Omron CX-Programmer project PAGODE (CX-Programmer 9.42)
; PLC1-GROND ; PLC2-GROND  ;PLC3-EILAND

# PLC PLC1_PAGODE: CS1G-H CPU42

## Global symbols (name address type ; comment)
ALM_1152_PLC2 H172.00 BOOL  ; ALARM PLC 2 WAARDE ACT-SOLL TE GROOT
ALM_EIL_BYPASS W226.15 BOOL  ; STAB EILAND IN BYPASS
ANA_OUT_2_REAL D5420 REAL  ; ANALOG OUTPUT 2 REAL 4-20mA
ANA_OUT_2_SCALER D5418 REAL  ; ANALOG OUTPUT 2 SCALER FOR 4-20mA
ARM_MOTION_PULSE 0142 NUMBER  ; ARM MOTION PULSER
ARM_POSITION_VALUE_ANA_OUT D5430 INT  ; ARM POSITION VALUE TO ANALOG OUTPUT
ARM_SPEED D5522 REAL  ; ARM SPEED IN DEGREE PER MINUTE
ARM_SPEED_FILTERED D6020 REAL  ; ARM SPEED FILTERED IN DEGREE PER MINUTE
ARM_SPEED_FILTER_01 D6000 REAL  ; ARM SPEED FILTER 01
ARM_SPEED_FILTER_02 D6002 REAL  ; ARM SPEED FILTER 01
ARM_SPEED_FILTER_03 D6004 REAL  ; ARM SPEED FILTER 03
ARM_SPEED_FILTER_04 D6006 REAL  ; ARM SPEED FILTER 04
ARM_SPEED_FILTER_05 D6008 REAL  ; ARM SPEED FILTER 05
ARM_SPEED_RESULT_01 D6010 REAL  ; RESULT 01
ARM_SPEED_RESULT_02 D6012 REAL  ; RESULT 02
ARM_SPEED_RESULT_03 D6014 REAL  ; RESULT 03
ARM_SPEED_RESULT_04 D6016 REAL  ; RESULT 04
Act_Snelheid_Aansturing_Arm D177 INT  ; Actuele snelheid aansturing Arm
1527.00 BOOL  ; Controllink Node 1 online
1527.01 BOOL  ; Controllink Node 2 online
1527.02 BOOL  ; Controllink Node 3 Online
2020.00 BOOL  ; COUNT
3012.02 BOOL  ; stop vanaf grond
3034.06 BOOL  ; COMMUNICATIE PLC 1 NAAR PLC 2 HYDRAULIEK UNIT ARM INBEDRIJF
3327.00 BOOL  ; Ingangspoort rechts gesloten Van PLC 2
3327.01 BOOL  ; Inganspoort links gesloten van PLC2
3337.03 BOOL  ; One Shot Pulse t.b.v. ramp tijd
56.05 BOOL  ; stop show
D1200 CHANNEL  ; SIMPLE COUNTER MODE
D1202 CHANNEL  ; COUNTER 2
D134 CHANNEL  ; help_abs_enc1
D190 CHANNEL  ; encoder_4_1
D191 CHANNEL  ; ecoder_4_2
D20 CHANNEL  ; `
H102.01 BOOL  ; Controllink Node 1 offline (PLC 1)
H102.02 BOOL  ; Controllink Node 2 offline (PLC 2)
H102.03 BOOL  ; Controllink Node 3 offline (PLC 3)
H102.05 BOOL  ; Algemene storing voor Controllink unit.
H102.06 BOOL  ; Storing Controllink Node 1
H102.07 BOOL  ; Storing Controllink Node 2
H102.08 BOOL  ; Storing Controllink Node 3
H121.03 BOOL  ; UPS in storing of batterijbedrijf
H121.04 BOOL  ; Alarm 1-0340 Hoge temperatuur in Technische Ruimte Pagode.
H158.09 BOOL  ; $?St$Bk?_#[29956] / Benedenpositie eiland wijkt af van encoder positie (42S10) / $?St$Bk?_#[29956]
H158.10 BOOL  ; $?St$Bk?_#[29957] / Ondermelding eiland niet binnen encoder waarden (41S4) / $?St$Bk?_#[29957]
H158.11 BOOL  ; $?St$Bk?_#[29958] / Ondermelding eiland niet binnen encoder waarden (41S7) / $?St$Bk?_#[29958]
H186.01 BOOL  ; $?St$Bk?_#[29959] / Alarm 1 - 1377 Poort 1 Links. Pal niet gevallen / $?St$Bk?_#[29959]
H186.02 BOOL  ; Alarm 1 - 1378 Poort 1 Links. Open sensor schakeld ongewenst. ( )
H186.03 BOOL  ; Alarm 1 - 1379 Poort 1 Links. Open sensor schakeld niet ( )
H186.04 BOOL  ; $?St$Bk?_#[29960] / Alarm 1 - 1380 Poort 1 Links. Bijna open sensor schakeld ongewenst. ( ) / $?St$Bk?_#[29960]
H186.05 BOOL  ; Alarm 1 - 1381 Poort 1 Links. Bijna open sensor schakeld niet ( )
H186.06 BOOL  ; Alarm 1 - 1382 Poort 1 Links. Sluit sensor schakeld ongewenst. ( )
H186.07 BOOL  ; Alarm 1 - 1383 Poort 1 Links. Sluit sensor schakeld niet ( )
H186.08 BOOL  ; $?St$Bk?_#[29961] / Alarm 1 - 1384 Poort 1 Links. Beknelling bewaking aangesproken. ( ) / $?St$Bk?_#[29961]
H400 CHANNEL  ; Algemene alarmen PLC 3 draaiend deel eiland
H401 CHANNEL  ; Alarmen Ingangspoort Links 1
H401.00 BOOL  ; $?St$Bk?_#[29962] / Alarm 1 - 1376 Poort 1 Links. Pal meldt niet omhoog / $?St$Bk?_#[29962]
H402 CHANNEL  ; Alarmen Ingangspoort Links 2
H403 CHANNEL  ; Alarmen Ingangspoort Rechts 1
H404 CHANNEL  ; Alarmen Ingangspoort Rechts 2
H405 CHANNEL  ; Alarmen Uitgangspoort Links 1
H406 CHANNEL  ; Alarmen Uitgangspoort Links 2
H407 CHANNEL  ; Alarmen Uitgangspoort Rechts 1
H408 CHANNEL  ; Alarmen Uitgangspoort Rechts 2
T0141 BOOL  ; DELAY ARM STAR
T0142 BOOL  ; ARM MOTION PULSER
T0150 BOOL  ; TIMER ENCODER 1 FAUT
T0151 BOOL  ; TIMER ENCODER 2 FAULT
T0198 BOOL  ; Delay Eiland op positie (1.04)
T0224 BOOL  ; ALARM 1-1454 SIGNAL STATUS VALVE 145 NOT OK
T0225 BOOL  ; ALARM 1-1455 OIL LEVEL 2 NOT OK
T0230 BOOL  ; ALARM 1-1462 HARDWARE WATCHDOG FROM HAGENBUCH MISSING TIMER ON
T0231 BOOL  ; ALARM 1-1462 HARDWARE WATCHDOG FROM HAGENBUCH MISSING TIMER OFF
T0240 BOOL  ; TIMER ARM HYDRAULIC ON
T0241 BOOL  ; TIMER ISLAND HYDRAULIC ON
T0310 BOOL  ; TIMER RESET ERROR HAGENBUCH SYSTEM
T0311 BOOL  ; PRESET INCLINOMETER HAGENBUCH
T0320 BOOL  ; Timer Alarm 1191
T0321 BOOL  ; Timer Alarm 1192
T0661 BOOL  ; \
W160.04 BOOL  ; blok_tourn
W160.06 BOOL  ; blokkeer_links
W160.07 BOOL  ; blokkeer_rechts
W20.03 BOOL  ; Merker Watchdog Communicatie OK Plc 1 & Plc 2
W231.15 BOOL  ; EILAND ROND GEWEEST
W56.03 BOOL  ; hydrau
W56.05 BOOL  ; stop show van grond
W56.06 BOOL  ; stop show van eiland
W90.00 BOOL  ; Blokkeer Tourniquet
W90.01 BOOL  ; Verhoog aantal
W90.02 BOOL  ; Blokkeer tourniquet links
W91.00 BOOL  ; Blokkeer Tourniquet
W91.01 BOOL  ; Verhoog aantal
W91.02 BOOL  ; Blokkeer tourniquet rechts
BT_Hydr_Main_Pump_Arm_On T0194 BOOL  ; Hydraulic main pump arm on delay timer
BT_MS_11Q08_not_OK T0195 BOOL  ; Hydraulic main pump arm MS 11Q08 not OK
BT_MS_11Q10_not_OK T0196 BOOL  ; Hydraulic main pump arm MS 11Q10 not OK
BT_MS_11Q12_not_OK T0197 BOOL  ; Hydraulic main pump arm MS 11Q12 not OK
COM1_AKTIEF_ALARM 3006.00 BOOL
COM1_ARM_ENAB_NEER 3024.03 BOOL  ; ARM ENABLE OMLAAG  VANUIT CYCLUS
COM1_ARM_OMHOOG 3037.00 BOOL  ; PLC 1 ARM OMHOOG
COM1_ARM_OMLAAG 3037.01 BOOL  ; PLC   1 ARM OMLAAG
COM1_ING_L_SLUITEN 3032.04 BOOL  ; VERZOEK SLUITEN INGANGS POORT LINKS
COM1_ING_R_OPEN 3032.05 BOOL  ; VERZOEK OPENEN INGANGS POORT RECHTS
COM1_ING_R_SLUITEN 3032.06 BOOL  ; VERZOEK SLUITEN INGANGS POORT RECHTS
COM1_Noodstop_Vertraagt_PLC1_OK 3004.04 BOOL  ; Communicatie Noodstop Vertaagt Plc 1 Ok Plc 1 naar Plc 2
COM1_STAPWOORD 3023 CHANNEL  ; STAP WOORD
COM1_TOURN_R 3031.01 BOOL  ; VERZOEK ENABLE TOURNIKET RECHTS
COM2_AKTIEF_ALARM 3306.00 BOOL
COM2_ARM_ENAB_NEER 3324.02 BOOL  ; ARM ENABLE OMLAAG VANUIT CYCLUS
COM2_ARM_ENAB_OP 3324.01 BOOL  ; ARM ENABLE OMHOOG VANUIT CYCLUS
COM2_ARM_OMHOOG 3337.00 BOOL  ; PLC 2 ARM OMHOOG
COM2_ARM_OMLAAG 3337.01 BOOL  ; PLC 2 ARM OMLAAG
COM2_ARM_SLOW 3324.05 BOOL  ; EILAND SLOW
COM2_CYCLUS_ENABLE 3324.15 BOOL  ; CYCLUS ENABLE
COM2_CYCLUS_STOP 3324.14 BOOL  ; VOORTIJDIGE STOP
COM2_EIL_STAB 3324.04 BOOL  ; EILAND STABILISATIE
COM2_ENAB_TOURNIKET 3324.10 BOOL  ; ENABLE TOURNIKET
COM2_ING_L_OPEN 3332.03 BOOL  ; VRIJGAVE INGANGS POORTEN L OPENEN VAN PLC 2
COM2_ING_L_SLUITEN 3332.04 BOOL  ; VRIJGAVE SLUITEN INGANGS POORT L VAN PLC 2
COM2_ING_R_OPEN 3332.05 BOOL  ; VRIJGAVE OPENEN INGANGS POORTEN RECHTS
COM2_ING_R_SLUITEN 3332.06 BOOL  ; VRIJGAVE SLUITEN INGANGS POORT RECHTS VAN PLC 2
COM2_LADING_WISSEL 3324.12 BOOL  ; BELADING EILAND WISSELEN
COM2_PB_EXIT_GATE 3033.00 BOOL  ; PUSH BUTTON EXIT GATE FROM ISLAND (PLC3)
COM2_POORT_DICHT 3324.09 BOOL  ; ALLE POORTEN GESLOTEN
COM2_POORT_ENAB 3324.00 BOOL  ; POORT ENABLE VANUIT CYCLUS
COM2_READY_START 3324.13 BOOL  ; READY VOOR START
COM2_RIDE_HOME 3324.11 BOOL  ; RIDE HOME
COM2_ROTATIE 3324.03 BOOL  ; ROTATIE ENABLE VANUIT CYCLUS
COM2_STAP0 3323.00 BOOL  ; STAP 0 CYCLUS
COM2_STAP1 3323.01 BOOL  ; STAP 1 CYCLUS
COM2_STAP10 3323.10 BOOL  ; STAP 10 CYCLUS
COM2_STAP13 3323.13 BOOL  ; STAP 13 CYCLUS
COM2_STAP14 3323.14 BOOL  ; STAP 14 CYCLUS
COM2_STAP15 3323.15 BOOL  ; STAP 15 CYCLUS
COM2_STAP2 3323.02 BOOL  ; STAP 2 CYCLUS
COM2_STAP3 3323.03 BOOL  ; STAP 3 CYCLUS
COM2_STAP4 3323.04 BOOL  ; STAP 4 CYCLUS
COM2_STAP5 3323.05 BOOL  ; STAP 5 CYCLUS
COM2_STAP6 3323.06 BOOL  ; STAP 6 CYCLUS
COM2_STAP7 3323.07 BOOL  ; STAP 7 CYCLUS
COM2_STAP8 3323.08 BOOL  ; STAP 8 CYCLUS
COM2_STAP9 3323.09 BOOL  ; STAP 9 CYCLUS
COM2_STAPWOORD 3323 CHANNEL  ; STAP WOORD
COM2_TOURN_L 3331.00 BOOL  ; TOESTEMMING VRIJG TOURNIKET L
COM2_TOURN_R 3331.01 BOOL  ; TOESTEMMING VRIGAVE TOURNIKET RECHTS
COM_TOURN_R 562.01 BOOL  ; VERZOEK VRIJGAVE TOURNIKET R
COUNTER_RESET_CH_1 2020.04 BOOL  ; COUNTER RESET CHANNEL 1
COUNTER_RESET_CH_2 2020.05 BOOL  ; COUNTER RESET CHANNEL 2
COUNT_CARD_CH1_INI D20201 CHANNEL  ; COUNTER CARD CHANNEL 1 INITIALISATION
COUNT_CARD_GEN_INI D20200 CHANNEL  ; COUNTER CARD GENERAL INITIALISATION
COUNT_GEN_ENABLE 2020.00 BOOL  ; COUNTERS GENERAL ENABLE
COUT_CARD_CH2_INI D20202 CHANNEL  ; COUNTER CARD CHANNEL 2 INITIALISATION
C_CONTROL D108 UINT  ; CONTROL BCD NAAR BIN COUNTERS
Com1_3_Eiland_Poortjes_Gesloten 906.00 BOOL  ; Merker Eiland Poortjes zijn Gesloten
Com1_3_Lamp_Ingangs_Poortjes_Geopend_Eiland 902.02 BOOL  ; Communicatie Lampje (16H2) Ingangs Poortje s 1 + 2 Geopend Eiland Plc 1 & Plc 2 naar Plc 3
Com1_3_Lamp_Ready_For_Dispatch 902.01 BOOL  ; Communicatie Ready for Dispatch Lampje Eiland (16H2) Plc 1 & Plc 2 naar Plc 3
Com1_3_Vrijgave_Poortjes_Eiland 906.01 BOOL  ; Communicatie Vrijgave Eiland Poortjes Plc 1 & Plc 2 naar Plc 3
Com1_44HS12 3011.15 BOOL
Com1_44HS14 3012.00 BOOL
Com1_91H10 3011.04 BOOL  ; Communicatie Lampje Algemeen Alarm Plc 1 naar Plc 2
Com1_91H12 3011.05 BOOL  ; Communicatie Lampje Show Plc 1 naar Plc 2
Com1_91H14 3011.06 BOOL  ; Communicatie Lampje Linkse Tourniquet Ontgrendelt Plc 1 naar Plc 2
Com1_91H16 3011.07 BOOL  ; Communicatie Lampje Rechtse Tourniquet Ontgrendelt Plc 1 naar Plc 2
Com1_91H18 3011.08 BOOL  ; Communicatie Lampje Arm & Eiland Omhoog Plc 1 naar Plc 2
Com1_91H2 3011.00 BOOL  ; Communicatie Lampje Sturrspanning Ingeschakeld Plc 1 naar Plc 2
Com1_91H4 3011.01 BOOL  ; Communicatei Lampje Handbedrijf Ingeschakeld Plc 1 naar Plc2
Com1_91H6 3011.02 BOOL  ; Communicatie Lampje Automatisch bedrijf Ingeschakeld Plc 1 naar Plc 2
Com1_91H8 3011.03 BOOL  ; Communicatie Lampje Pompen in Bedrijf Plc 1 naar Plc 2
Com1_92H12 3011.14 BOOL
Com1_92H2 3011.09 BOOL  ; Communicatie Lampje Arm & Eiland Omlaag Plc 1 naar Plc 2
Com1_92H4 3011.10 BOOL  ; Communicatie Lampje Rotatie Eiland Linksom Plc 1 naar Plc 2
Com1_92H6 3011.11 BOOL  ; Communicatie Lampje Rotatie Eiland Rechtsom Plc 1 naar Plc 2
Com1_92H8 3011.12 BOOL  ; Service schakelaar technische dients
Com1_92S14 3011.15 BOOL
Com1_92Z10 3011.13 BOOL
Com1_Act_Groter_Snelheid 3037.04 BOOL  ; Actuele snelheid groter dan wens snelheid
Com1_Act_Kleiner_Snelheid 3037.06 BOOL  ; Actuele snelheid kleiner dan wens snelheid
Com1_Act_gelijk_Snelheid 3037.05 BOOL  ; Actuele snelheid gelijk aan de wens snelheid
Com1_Arm_Home 3024.01 BOOL  ; Arm is geheel beneden
Com1_Arm_Omhoog 3037.01 BOOL  ; PLC 1 ARM OMHOOG
Com1_Arm_Omlaag 3037.02 BOOL  ; PLC 1ARM OMLAAG
Com1_Auto_Bedrijf 3010.01 BOOL  ; Communicatie Auto Bedrijf van Plc 1 Naar Plc 2
Com1_Auto_Rotatie_Rechtsom 3047.02 BOOL
Com1_Auto_Rotatie_linksom 3047.01 BOOL  ; Communicatie Auto Rotatie Linksom
Com1_E_Stop_Niet_Gedrukt 3004.00 BOOL  ; Communicatie E-stop niet gedrukt Plc 1 naar Plc 2
Com1_Eiland_Poortjes_Gesloten 3044.00 BOOL  ; Communicatie Eiland Poortjes Gesloten Plc 1 naar Plc 2
Com1_Eiland_Rond_Geweest 3047.14 BOOL
Com1_Eiland_Stab_Linksom 3046.01 BOOL  ; Communicatie Plc 1 naar Plc 2 Stabiliseer het Eiland naar Links
Com1_Eiland_Stab_Rechtsom 3046.02 BOOL  ; Communicatie Plc 1 naar Plc 2 Stabiliseer het Eiland naar Rechts
Com1_Enable_Freq_Contr_Linksom 3047.13 BOOL
Com1_Enable_Freq_Contr_Rechtsom 3047.12 BOOL
Com1_Enable_Hydrau_Eiland 3045.00 BOOL  ; Communicatie Enable Hydrau Eiland Plc 1 naar Plc 2
Com1_Enable_Stabilisatie 3046.00 BOOL  ; Communicatie Plc 1 naar Plc 2 Enable de Eiland Stabilisatie
Com1_Hand_Bedrijf 3010.00 BOOL  ; Communicatie Hand Bedrijf Plc 1 naar plc 2
Com1_Hardw_Watchdogs_OK 3003.05 BOOL  ; Communicatie Plc 1 Watchdog plc 2 ok
Com1_Hardw_Watchdogs_ON 3003.04 BOOL  ; Communicatie Hardware Watchdog Plc 1 ON
Com1_Hoofd_Pomp_Hydrau_Grond 3034.02 BOOL  ; COMMUNICATIE PLC 1 NAAR PLC 2 START HOOFDPOMP HYDRAULIEK UNIT ARM
Com1_Hoofdpomp_Hydrau_Eiland 3045.03 BOOL  ; Communicatie Hoofdmotor Hydrau Eiland Aan Plc 1 naar Plc 2
Com1_Hoofdschakelaar_OK 3008.01 BOOL  ; Communicatie Hoofdschakelaar (3K7) OK (geen Kortsluiting of overbelasting)
Com1_Hydrau_Arm_OK 3034.06 BOOL  ; COMMUNICATIE PLC 1 NAAR PLC 2 HYDRAULIEK UNIT ARM INBEDRIJF
Com1_Hydrau_Eiland_ON 3045.01 BOOL  ; Communicatie Start Hydrau Pompen Plc 1 naar Plc 2
Com1_Hydrauliek_Eiland_Inbedrijf 3045.15 BOOL
Com1_Ingang_Poortje_1_L_Dicht 3032.02 BOOL  ; Communicatie Plc 1 naar Plc 2 Open Ingangs poortjes
Com1_Ingangs_Poortje_1_Links_Open 3032.01 BOOL
Com1_Ingangs_Poortjes_Gesloten 3032.07 BOOL
Com1_Inst_Autom_7F12_Eiland_OK 3008.13 BOOL  ; Communicatie Installatie-Automaat Eiland (7F12) OK Plc 1 naar Plc 2
Com1_Inst_Autom_7F3_Eiland_OK 3008.10 BOOL  ; Communicatie Installatie-Automaat Eiland (7F3) OK Plc 1 naar Plc 2
Com1_Inst_Autom_7F5_Eiland_OK 3008.11 BOOL  ; Communicatie Installatie-Automaat Eiland (7F5) OK Plc 1 naar Plc 2
Com1_Inst_Autom_7F7_Eiland_OK 3008.12 BOOL  ; Communicatie Installatie-Automaat Eiland (7F7) OK Plc 1 naar Plc 2
Com1_Inst_Autom_8F11_Eiland_OK 3008.15 BOOL  ; Communicatie Installatie-Automaat Eiland (8F11) OK Plc 1 naar Plc 2
Com1_Inst_Autom_8F14_Eiland_OK 3009.00 BOOL  ; Communicatie Installatie-Automaat Eiland (8F14) OK Plc 1 naar Plc 2
Com1_Inst_Autom_8F17_Eiland_OK 3009.01 BOOL  ; Communicatie Installatie-Automaat Eiland (8F17) OK Plc 1 naar Plc 2
Com1_Inst_Autom_8F3_Eiland_OK 3008.14 BOOL  ; Communicatie Installatie-Automaat Eiland (8F3) OK Plc 1 naar Plc 2
Com1_Inst_Automaat_7F3_OK 3008.02 BOOL  ; Communicatie Installatie-Automaat (7F3) OK Plc 1 naar Plc 2
Com1_Inst_Automaat_7F5_OK 3008.03 BOOL  ; Communicatie Installatie-Automaat (7F5) OK Plc 1 naar Plc 2
Com1_Inst_Automaat_7F7_OK 3008.04 BOOL  ; Communicatie Installatie-Automaat (7F7) OK Plc 1 naar Plc 2
Com1_Inst_Automaat_8F11_OK 3008.06 BOOL  ; Communicatie Installatie-Automaat (8F11) OK Plc 1 naar Plc 2
Com1_Inst_Automaat_8F13_OK 3008.07 BOOL  ; Communicatie Installatie-Automaat (8F13) OK Plc 1 naar Plc 2
Com1_Inst_Automaat_8F15_OK 3008.08 BOOL  ; Communicatie Installatie-Automaat (8F15) OK Plc 1 naar Plc 2
Com1_Inst_Automaat_8F3_OK 3008.05 BOOL  ; Communicatie Installatie-Automaat (8F3) OK Plc 1 naar Plc 2
Com1_Inst_Automaat_9F11_OK 3008.09 BOOL  ; Communicatie Installatie-Automaat (9F11) OK Plc 1 naar Plc 2
Com1_Koelingspomp_Hydrau_Arm 3034.03 BOOL  ; COMMUNICATIE PLC 1 NAAR PLC 2 START KOELER POMP HYDRAULIEK UNIT ARM
Com1_Lamp_Eiland_Ingangs_poortjes_Geopend 3013.02 BOOL  ; Communicatie Lampje (16H2) Ingangs Poortje s 1 + 2 Geopend Eiland Plc 1 naar Plc 2
Com1_Lamp_Eiland_Ingangs_poortjes_Gesloten 3013.03 BOOL  ; Communicatie Lampje (16H3) Ingangs Poortje s 1 + 2 Gesloten Eiland Plc 1 naar Plc 2
Com1_Lamp_Eiland_Uitgangs_poortjes_Geopend 3013.05 BOOL  ; Communicatie Lampje (16H4) Uitgangs Poortje s 1 + 2 Geopend Eiland Plc 1 naar Plc 2
Com1_Lamp_Ready_For_Dispatch 3013.01 BOOL  ; Communicatie Lampje (16H3) Ready For Dispatch Eiland Plc 1 naar Plc 2
Com1_Noodstop_Direct_PLC1_OK 3004.03 BOOL  ; Communicatie NoodStop Direct OK Plc 1 naar Plc 2
Com1_Noodstop_PLC_1_OK 3004.02 BOOL  ; Communicatie Noodstop Plc 1 OK
Com1_Open_Ingangs_Poort_1_L 3032.03 BOOL
Com1_Open_Uitgangs_Poortjes 3033.03 BOOL  ; Open de Uitgangs Poortjes
Com1_Power_Freq_Reg_4A1 3047.00 BOOL  ; Communicatie Frequentie Regelaar (4A1) Voeding (72K6) Plc 1 naar 2
Com1_Pulse 3037.03 BOOL
Com1_Ready_To_Start_Show 3024.07 BOOL  ; Ready to Start Show
Com1_Ready_to_Reset_E_Stop 3004.01 BOOL  ; Communicatie Ready om de Noodstop te Resetten Plc 1 naar Plc 2
Com1_Reinigingspomp_Hydrau_Arm 3034.04 BOOL  ; COMMUNICATIE PLC 1 NAAR PLC 2 START OLIE REINIGINGS POMP HYDRAULIEK UNIT ARM
Com1_Reset_Trigger 3037.07 BOOL
Com1_Rotatie_Linksom 3047.04 BOOL
Com1_Rotatie_Rechtsom 3047.08 BOOL
Com1_Rotatie_Snel_Linksom 3047.06 BOOL
Com1_Rotatie_Snel_Rechtsom 3047.10 BOOL
Com1_Rotatie_Traag_Linksom 3047.05 BOOL
Com1_Rotatie_Traag_Rechtsom 3047.09 BOOL
Com1_SK_Open_Linker_Ingangs_Poortje_Eiland 3014.09 BOOL
Com1_SK_Open_Linker_Ingangs_Poortje_Oever 3014.11 BOOL
Com1_SK_Open_Linker_Uitgangs_Poortjes_Eiland 3014.13 BOOL
Com1_SK_Open_Rechter_Ingangs_Poortje_Eiland 3014.10 BOOL
Com1_SK_Open_Rechter_Ingangs_Poortje_Oever 3014.12 BOOL
Com1_SK_Open_Rechter_Uitgangs_Poortje_Eiland 3014.14 BOOL
Com1_SK_Open_Sluit_Linker_Oever_Poortjes_ 3014.05 BOOL
Com1_SK_Open_Sluit_Rechter_Oever_Poortjes_ 3014.06 BOOL
Com1_SK_Open_Uitgangs_Poortjes_Oever 3014.15 BOOL
Com1_SK_Reset_Alarmen 3014.01 BOOL
Com1_SK_SPARE_3314_00 3014.00 BOOL
Com1_SK_SPARE_3314_02 3014.02 BOOL
Com1_SK_SPARE_3315_03 3015.02 BOOL
Com1_SK_SPARE_3315_07 3015.07 BOOL
Com1_SK_SPARE_3315_08 3015.08 BOOL
Com1_SK_SPARE_3315_09 3015.09 BOOL
Com1_SK_Stabilisatie_Eiland_Linksom 3015.05 BOOL
Com1_SK_Stabilisatie_Eiland_Rechtsom 3015.06 BOOL
Com1_SK_Start_Stop_Hoofdpomp_Arm 3015.01 BOOL
Com1_SK_Start_Stop_Hoofdpomp_Eiland 3015.04 BOOL
Com1_SK_Start_Stop_Hydrau 3014.03 BOOL
Com1_SK_Start_Stop_Show 3014.04 BOOL
Com1_SK_Start_Stop_Stuurpomp_Arm 3015.00 BOOL
Com1_SK_Start_Stop_Stuurpomp_Eiland 3015.03 BOOL
Com1_SK_Vrijgave_Linker_Tourniquet 3014.07 BOOL
Com1_SK_Vrijgave_Rechter_Tourniquet 3014.08 BOOL
Com1_SK_WCD_1 3015.10 BOOL
Com1_SK_WCD_2 3015.11 BOOL
Com1_SK_WCD_3 3015.12 BOOL
Com1_SK_WCD_4 3015.13 BOOL
Com1_SK_WCD_5 3015.14 BOOL
Com1_SK_WCD_6 3015.15 BOOL
Com1_Service_Bedrijf_Ch_A 3010.02 BOOL  ; Communicatie Service Bedrijf Channel A van Plc 1 Naar Plc 2
Com1_Service_Bedrijf_Ch_B 3010.03 BOOL  ; Communicatie Service Bedrijf Channel B van Plc 1 Naar Plc 2
Com1_Show_Afbreken 3024.04 BOOL  ; Show Afbreken
Com1_Show_Arm_Omhoog 3024.08 BOOL  ; Show Arm Omhoog
Com1_Show_Arm_Omlaag 3024.09 BOOL  ; Show Arm Omlaag
Com1_Show_Eiland_Rotatie 3024.11 BOOL  ; Show Eiland Rotatie
Com1_Show_Eiland_Stabilisatie 3024.10 BOOL  ; Show Eiland Stabilisatie
Com1_Show_Stap_0 3023.00 BOOL  ; Show Stap 0
Com1_Show_Stap_1 3023.01 BOOL  ; Show Stap 1
Com1_Show_Stap_10 3023.10 BOOL  ; Show Stap 10
Com1_Show_Stap_2 3023.02 BOOL  ; Show Stap 2
Com1_Show_Stap_4 3023.04 BOOL  ; Show Stap 4
Com1_Show_Stap_5 3023.05 BOOL  ; Show Stap 5
Com1_Show_Stap_6 3023.06 BOOL  ; Show Stap 6
Com1_Show_Stap_7 3023.07 BOOL  ; Show Stap 7
Com1_Show_Stap_8A 3023.11 BOOL  ; Show Stap 8 A
Com1_Show_Stap_8B 3023.12 BOOL  ; Show Stap 8 B
Com1_Show_Stap_9 3023.09 BOOL  ; Show Stap 9
Com1_Show_stap_8 3023.08 BOOL  ; Show Stap 8
Com1_Sluit_Uitgangs_Poortjes_Oever 3033.04 BOOL  ; Sluit de Uitgangs Poortjes Oever
Com1_Smeertoestel_Hydrau_Arm 3034.05 BOOL  ; COMMUNICATIE PLC 1 NAAR PLC 2 START SMEER TOESTEL HYDRAULIEK UNIT ARM
Com1_Softw_Watchdog_Plc_2_OK 3003.03 BOOL  ; Communicatie Software Watchdog Plc 2 OK
Com1_Softw_watchdog_Plc_1_on 3003.00 BOOL  ; Communicatie Plc 1 Watchdog plc 1 on
Com1_Softw_watchdog_Pulse_Plc_1 3003.01 BOOL  ; Communicatie Software Watchdog Pulse Plc 1
Com1_Spannings_Beveiliging_OK 3008.00 BOOL  ; Communicatie Onder- OverSpannings beveiliging OK
Com1_Stap_3 3023.03 BOOL  ; Show Stap 3
Com1_Stop_Show 3024.05 BOOL  ; Stop Show
Com1_Stuur_Pomp_Hydrau_Grond 3034.01 BOOL  ; VERZOEK  STUUR POMP HYDRAULIEK UNIT ARM
Com1_Stuurpomp_Hydrau_Arm 3034.01 BOOL  ; COMMUNICATIE PLC 1 NAAR PLC 2 START STUUR POMP HYDRAULIEK UNIT ARM
Com1_Stuurpomp_Hydrau_Eiland 3045.02 BOOL  ; Communicatie StuurPompen Aan Hydrualiek Eiland Plc 1 naar Plc 2
Com1_Tilt_switches_OK 3042.00 BOOL  ; Communicatie Tilt Switches OK Plc 1 naar Plc 2
Com1_Uitgangs_poortjes_Dicht 3033.02 BOOL  ; Uitgangs Poortjes zijn Gesloten
Com1_Uitgangs_poortjes_Open 3033.01 BOOL  ; Uitgangs Poortjes Zijn Open
Com1_VRIJGAVE_HYDRAU_ARM 3034.00 BOOL  ; COMMUNICATIE PLC 1 NAAR PLC 2 VRIJGAVE HYDRAULIEK UNIT ARM
Com1_Verhinder_Start_Show 3024.06 BOOL  ; Verhinder de Start van de Show
Com1_Vrijgave_Arm_Beweging 3037.00 BOOL
Com1_Vrijgave_Eiland_Poortjes 3044.01 BOOL  ; Communicatie Vrijgave Eiland Poortjes Plc 1 naar Plc 2
Com1_Vrijgave_Ingangs_Poortjes 3032.00 BOOL
Com1_Vrijgave_L_Tourniket 3031.00 BOOL  ; Communicatie Plc 1 Naar Plc 2 Vrijgave Linker Tourniquets
Com1_Vrijgave_Poortjes_OK 3021.00 BOOL  ; Communicatie Vrijgave Poortjes OK Plc 1 naar Plc 2
Com1_Vrijgave_Rem_1_2_3_4 3047.11 BOOL
Com1_Vrijgave_Rotatie_Rechtsom 3047.07 BOOL
Com1_Vrijgave_Rotatie_linksom 3047.03 BOOL
Com1_Vrijgave_Show 3024.00 BOOL
Com1_Vrijgave_Tourniquets 3021.01 BOOL  ; communicatie Vrijgave Tourniquets OK Plc 1 naar Plc 2
Com2_44HS12 3311.15 BOOL
Com2_44HS14 3312.00 BOOL
Com2_91H10 3311.05 BOOL  ; Communicatie Lampje Algemeen Alarm Plc 2 naar Plc 1
Com2_91H12 3311.06 BOOL  ; Communicatie Lampje Show Plc 2 naar Plc 1
Com2_91H14 3311.07 BOOL  ; Communicatie Lampje Linkse Tourniquet Ontgrendelt Plc 2 naar Plc 1
Com2_91H16 3311.08 BOOL  ; Communicatie Lampje Rechtse Tourniquet Ontgrendelt Plc 2 naar Plc 1
Com2_91H18 3311.09 BOOL  ; Communicatie Lampje Arm & Eiland Omhoog Plc 2 naar Plc 1
Com2_91H2 3311.01 BOOL  ; Communicatie Lampje Sturrspanning Ingeschakeld Plc 2 naar Plc 1
Com2_91H4 3311.02 BOOL  ; Communicatei Lampje Handbedrijf Ingeschakeld Plc 2 naar Plc 1
Com2_91H6 3311.03 BOOL  ; Communicatie Lampje Automatisch bedrijf Ingeschakeld Plc 2 naar Plc 1
Com2_91H8 3311.04 BOOL  ; Communicatie Lampje Pompen in Bedrijf Plc 2 naar Plc 1
Com2_92H2 3311.10 BOOL  ; Communicatie Lampje Arm & Eiland Omlaag Plc 2 naar Plc 1
Com2_92H4 3311.11 BOOL  ; Communicatie Lampje Rotatie Eiland Linksom Plc 2 naar Plc 1
Com2_92H6 3311.12 BOOL  ; Communicatie Lampje Rotatie Eiland Linksom Plc 2 naar Plc 1
Com2_Act_Groter_Snelheid 3337.04 BOOL  ; Actuele snelheid groter dan wens snelheid
Com2_Act_Kleiner_Snelheid 3337.06 BOOL  ; Actuele snelheid kleiner dan wens snelheid
Com2_Act_gelijk_Snelheid 3337.05 BOOL  ; Actuele snelheid gelijk aan de wens snelheid
Com2_Arm_Home 3324.01 BOOL  ; Arm is geheel beneden
Com2_Arm_Omhoog 3337.01 BOOL  ; PLC 2 ARM OMHOOG
Com2_Arm_Omlaag 3337.02 BOOL  ; PLC 2 ARM OMLAAG
Com2_Auto_Bedrijf 3310.01 BOOL  ; Communicatie Auto Bedrijf van Plc 2 Naar Plc 1
Com2_Auto_Rotatie_Rechtsom 3347.02 BOOL
Com2_Auto_Rotatie_linksom 3347.01 BOOL
Com2_E_Stop_Niet_Gedrukt 3304.00 BOOL  ; Communicatie E-stop niet gedrukt Plc 2
Com2_Eiland_Home 3324.02 BOOL  ; Het Eiland Is geheel Links- of Rechtsom Gedraaid
Com2_Eiland_Poortjes_Gesloten 3344.00 BOOL  ; Communicatie Eiland Poortjes Gesloten Plc 2 naar Plc 1
Com2_Eiland_Rond_Geweest 3347.14 BOOL
Com2_Eiland_Stab_Linksom 3346.01 BOOL
Com2_Eiland_Stab_Rechtsom 3346.02 BOOL  ; Communicatie Plc 2 naar Plc 1 Stabiliseer het Eiland naar Rechts
Com2_Enable_Freq_Contr_Linksom 3347.13 BOOL
Com2_Enable_Freq_Contr_Rechtsom 3347.12 BOOL
Com2_Enable_Hydrau_Eiland 3345.00 BOOL  ; Communicatie Enable Hydrau Eiland Plc 2 naar Plc 1
Com2_Enable_Stabilisatie 3346.00 BOOL
Com2_HOOFD_HYDRAU_EIL 3345.01 BOOL  ; VRIJGAVE PLC 2 HOOFDPOMP EILAND
Com2_Hand_Bedrijf 3310.00 BOOL  ; Communicatie Hand Bedrijf Plc 2 naar plc 1
Com2_Hardw_Watchdogs_OK 3300.04 BOOL  ; Communicatie Plc 2 Watchdog plc 1 ok
Com2_Hardw_Watchdogs_ON 3303.04 BOOL  ; Communicatie Hardware Watchdog Plc 2 ON
Com2_Hoofd_Pomp_Hydrau_Grond 3334.02 BOOL  ; COMMUNICATIE PLC 2 NAAR PLC 1 START HOOFD POMP HYDRAULIEK UNIT ARM
Com2_Hoofdpomp_Hydrau_Eiland 3345.03 BOOL  ; Communicatie Hoofdmotor Hydrau Eiland Aan Plc 2 naar Plc 1
Com2_Hoofdschakelaar_OK 3308.01 BOOL  ; Communicatie Hoofdschakelaar (3K7) OK (geen Kortsluiting of overbelasting) Plc 2 naar Plc 1
Com2_Hydrau_Arm_OK 3334.06 BOOL  ; COMMUNICATIE PLC 2 NAAR PLC 1 HYDRAULIEK UNIT ARM INBEDRIJF
Com2_Hydrau_Eiland_ON 3345.01 BOOL  ; Communicatie Start Hydrau Pompen Plc 2 naar Plc 1
Com2_Hydrauliek_Eiland_Inbedrijf 3345.15 BOOL
Com2_Ingangs_Poortje_1_L_Dicht 3332.02 BOOL  ; Communicatie Plc 2 naar Plc 1 Open Ingangs poortjes
Com2_Ingangs_Poortje_1_Links_Open 3332.01 BOOL
Com2_Ingangs_Poortjes_Gesloten 3332.07 BOOL
Com2_Input_0_00 3375.00 BOOL  ; Com2_Input_0_00
Com2_Inst_Autom_7F12_Eiland_OK 3308.13 BOOL  ; Communicatie Installatie-Automaat Eiland (7F12) OK Plc 2 naar Plc 1
Com2_Inst_Autom_7F3_Eiland_OK 3308.10 BOOL
Com2_Inst_Autom_7F5_Eiland_OK 3308.11 BOOL  ; Communicatie Installatie-Automaat Eiland (7F5) OK Plc 2 naar Plc 1
Com2_Inst_Autom_7F7_Eiland_OK 3308.12 BOOL  ; Communicatie Installatie-Automaat Eiland (7F7) OK Plc 2 naar Plc 1
Com2_Inst_Autom_8F11_Eiland_OK 3308.15 BOOL  ; Communicatie Installatie-Automaat Eiland (8F11) OK Plc 2 naar Plc 1
Com2_Inst_Autom_8F14_Eiland_OK 3309.00 BOOL  ; Communicatie Installatie-Automaat Eiland (8F14) OK Plc 2 naar Plc 1
Com2_Inst_Autom_8F17_Eiland_OK 3309.01 BOOL  ; Communicatie Installatie-Automaat Eiland (8F17) OK Plc 2 naar Plc 1
Com2_Inst_Autom_8F3_Eiland_OK 3308.14 BOOL  ; Communicatie Installatie-Automaat Eiland (8F3) OK Plc 2 naar Plc 1
Com2_Inst_Automaat_7F3_OK 3308.02 BOOL  ; Communicatie Installatie-Automaat (7F3) OK Plc 2 naar Plc 1
Com2_Inst_Automaat_7F5_OK 3308.03 BOOL  ; Communicatie Installatie-Automaat (7F5) OK Plc 2 naar Plc 1
Com2_Inst_Automaat_7F7_OK 3308.04 BOOL  ; Communicatie Installatie-Automaat (7F7) OK Plc 2 naar Plc 1
Com2_Inst_Automaat_8F11_OK 3308.06 BOOL  ; Communicatie Installatie-Automaat (8F11) OK Plc 2 naar Plc 1
Com2_Inst_Automaat_8F13_OK 3308.07 BOOL  ; Communicatie Installatie-Automaat (8F13) OK Plc 2 naar Plc 1
Com2_Inst_Automaat_8F15_OK 3308.08 BOOL  ; Communicatie Installatie-Automaat (8F15) OK Plc 2 naar Plc 1
Com2_Inst_Automaat_8F3_OK 3308.05 BOOL  ; Communicatie Installatie-Automaat (8F3) OK Plc 2 naar Plc 1
Com2_Inst_Automaat_9F11_OK 3308.09 BOOL  ; Communicatie Installatie-Automaat (9F11) OK Plc 2 naar Plc 1
Com2_Lamp_Eiland_Ingangs_poortjes_Geopend 3313.02 BOOL  ; Communicatie Lampje (16H2) Ingangs Poortje s 1 + 2 Geopend Eiland Plc 2 naar Plc 1
Com2_Lamp_Eiland_Ingangs_poortjes_Gesloten 3313.03 BOOL  ; Communicatie Lampje (16H3) Ingangs Poortje s 1 + 2 Gesloten Eiland Plc 2 naar Plc 1
Com2_Lamp_Ready_For_Dispatch 3313.01 BOOL  ; Communicatie Lampje (16H1) Ready For Dispatch Eiland Plc 2 naar Plc 1
Com2_Noodstop_Direct_PLC2_OK 3304.03 BOOL  ; Communicatie NoodStop Direct OK Plc 2 naar Plc 1
Com2_Noodstop_PLC_2_OK 3304.02 BOOL  ; Communicatie NoodStop Plc 2 OK
Com2_Noodstop_Vertraagt_PLC2_OK 3304.04 BOOL  ; Communicatie Noodstop Vertaagt Plc 2 Ok Plc 2 naar Plc 1
Com2_Open_Uitgangs_Poortjes 3333.03 BOOL  ; Open de Uitgangs Poortjes
Com2_Poortjes_Gesloten 3324.03 BOOL  ; Alle Oever & Eiland Poortjes zijn Gesloten
Com2_Power_Freq_Reg_4A1 3347.00 BOOL  ; Communicatie Frequentie Regelaar (4A1) Voeding (72K6) Plc 2 naar 1
Com2_Ready_To_Start_Show 3324.07 BOOL  ; Ready to Start Show
Com2_Ready_to_Reset_E_STOP 3304.01 BOOL  ; Communicatie Plc 2 is Ready om de Noodstop te Resetten
Com2_Reinigingspomp_Hydrau_Arm 3334.04 BOOL  ; COMMUNICATIE PLC 2 NAAR PLC 1 START OLIE REINIGINGS POMP HYDRAULIEK UNIT ARM
Com2_Rinigingspomp_Hydrau_Arm 3334.03 BOOL  ; COMMUNICATIE PLC 2 NAAR PLC 1  START KOELER POMP HYDRAULIEK UNIT ARM
Com2_Rotatie_Linksom 3347.04 BOOL
Com2_Rotatie_Rechtsom 3347.08 BOOL
Com2_Rotatie_Snel_Linksom 3347.06 BOOL
Com2_Rotatie_Snel_Rechtsom 3347.10 BOOL
Com2_Rotatie_Traag_Linksom 3347.05 BOOL
Com2_Rotatie_Traag_Rechtsom 3347.09 BOOL
Com2_SK_Open_Linker_Ingangs_Poortje_Eiland 3314.09 BOOL  ; Skada Bediening Open Linker Ingangs Poortje Eiland
Com2_SK_Open_Linker_Ingangs_Poortje_Oever 3314.11 BOOL  ; Skada Bediening Open Linker Ingangs Poortje Oever
Com2_SK_Open_Linker_Uitgangs_Poortjes_Eiland 3314.13 BOOL  ; Skada Bediening Open Linker Uitgangs Poortje Eiland
Com2_SK_Open_Rechter_Ingangs_Poortje_Eiland 3314.10 BOOL  ; Skada Bediening Open Rechter ingangs poortje Eiland
Com2_SK_Open_Rechter_Ingangs_Poortje_Oever 3314.12 BOOL  ; Skada Bediening Open Rechter ingangs poortje Oever
Com2_SK_Open_Rechter_Uitgangs_Poortje_Eiland 3314.14 BOOL  ; Skada Bediening Open Rechter Uitgangs poortje Eiland
Com2_SK_Open_Sluit_Linker_Oever_Poortjes_ 3314.05 BOOL  ; Skada Bediening Open / Sluit Linker Oever Poortjes
Com2_SK_Open_Sluit_Rechter_Oever_Poortjes_ 3314.06 BOOL  ; Skada Bediening Open / Sluit Rechter Oever Poortjes
Com2_SK_Open_Uitgangs_Poortjes_Oever 3314.15 BOOL  ; Skada Bediening Open Uitgangs poortjes Oever
Com2_SK_Reset_Alarmen 3314.01 BOOL  ; Skada Bediening Reset Alarmen
Com2_SK_SPARE_3314_00 3314.00 BOOL
Com2_SK_SPARE_3314_02 3314.02 BOOL
Com2_SK_SPARE_3315_03 3315.02 BOOL
Com2_SK_SPARE_3315_07 3315.07 BOOL
Com2_SK_SPARE_3315_08 3315.08 BOOL
Com2_SK_SPARE_3315_09 3315.09 BOOL
Com2_SK_Stabilisatie_Eiland_Linksom 3315.05 BOOL  ; Skada Bediening Eiland Stabilisatie Linksom
Com2_SK_Stabilisatie_Eiland_Rechtsom 3315.06 BOOL  ; Skada Bediening Eiland Stabilisatie Rechtsom
Com2_SK_Start_Stop_Hoofdpomp_Arm 3315.01 BOOL  ; Skada Bediening Start / Stop Hydrauliek Hoofdpomp Arm
Com2_SK_Start_Stop_Hoofdpomp_Eiland 3315.04 BOOL  ; Skada Bediening Start / Stop Hydrauliek Hoofdpomp Eiland
Com2_SK_Start_Stop_Hydrau 3314.03 BOOL  ; Skada Bediening Start / Stop Hydrauliek Arm & Eiland
Com2_SK_Start_Stop_Show 3314.04 BOOL  ; Skada Bediening Start / Stop Show
Com2_SK_Start_Stop_Stuurpomp_Arm 3315.00 BOOL  ; Skada Bediening Start / Stop Hydrauliek Stuurpomp Arm
Com2_SK_Start_Stop_Stuurpomp_Eiland 3315.03 BOOL  ; Skada Bediening Start / Stop Hydrauliek Stuurpomp Eiland
Com2_SK_Vrijgave_Linker_Tourniquet 3314.07 BOOL  ; Skada bediening Vrijgave Linker Tourniquets
Com2_SK_Vrijgave_Rechter_Tourniquet 3314.08 BOOL  ; Skada Bediening Vrijgave Rechter Tourniquets
Com2_SK_WCD_1 3315.10 BOOL  ; Skada Bediening Wandcontactdoos 1
Com2_SK_WCD_2 3315.11 BOOL  ; Skada Bediening Wandcontactdoos 2
Com2_SK_WCD_3 3315.12 BOOL  ; Skada Bediening Wandcontactdoos 3
Com2_SK_WCD_4 3315.13 BOOL  ; Skada Bediening Wandcontactdoos 4
Com2_SK_WCD_5 3315.14 BOOL  ; Skada Bediening Wandcontactdoos 5
Com2_SK_WCD_6 3315.15 BOOL  ; Skada Bediening Wandcontactdoos 6
Com2_SPANNINGS_BEVEILIGING_OK 3308.00 BOOL  ; Communicatie Onder- OverSpannings beveiliging OK
Com2_Service_Bedrijf_Ch_A 3310.02 BOOL  ; Communicatie Service Bedrijf van Plc 2 Naar Plc 1 Channel A
Com2_Service_Bedrijf_Ch_B 3310.03 BOOL  ; Communicatie Service Bedrijf van Plc 2 Naar Plc 1 Channel B
Com2_Show_Afbreken 3324.04 BOOL  ; Show Afbreken
Com2_Show_Arm_Omhoog 3324.08 BOOL  ; Show Arm Omhoog
Com2_Show_Arm_Omlaag 3324.09 BOOL  ; Show Arm Omlaag
Com2_Show_Eiland_Rotatie 3324.11 BOOL  ; Show Eiland Rotatie
Com2_Show_Eiland_Stabilisatie 3324.10 BOOL  ; Show Eiland Stabilisatie
Com2_Show_Stap_0 3323.00 BOOL  ; Show Stap 0
Com2_Show_Stap_1 3323.01 BOOL  ; Show Stap 1
Com2_Show_Stap_10 3323.10 BOOL  ; Show Stap 10
Com2_Show_Stap_2 3323.02 BOOL  ; Show Stap 2
Com2_Show_Stap_3 3323.03 BOOL  ; Show Stap 3
Com2_Show_Stap_4 3323.04 BOOL  ; Show Stap 4
Com2_Show_Stap_5 3323.05 BOOL  ; Show _Stap_5
Com2_Show_Stap_6 3323.06 BOOL  ; Show Stap 6
Com2_Show_Stap_7 3323.07 BOOL  ; Show Stap 7
Com2_Show_Stap_8 3323.08 BOOL  ; Show Stap 8
Com2_Show_Stap_8A 3323.11 BOOL  ; Show Stap 8 A
Com2_Show_Stap_8B 3323.12 BOOL  ; Show Stap 8 B
Com2_Show_Stap_9 3323.09 BOOL  ; Show Stap 9
Com2_Sluit_Uitgangs_Poortjes_Oever 3333.04 BOOL  ; Sluit de Uitgangs Poortjes Oever
Com2_Smeertoestel_Hydrau_Arm 3334.05 BOOL  ; COMMUNICATIE PLC 2 NAAR PLC 1 START SMEER TOESTEL HYDRAULIEK UNIT ARM
Com2_Softw_Watchdog_Plc_1_OK 3303.03 BOOL  ; Communicatie Software Watchdog Plc 1 OK
Com2_Softw_watchdog_Plc_2_on 3303.00 BOOL  ; Communicatie Plc 2 Watchdog plc 1 on
Com2_Softw_watchdog_Pulse_Plc_2 3303.01 BOOL  ; Communicatie Software Watchdog Pulse Plc 2
Com2_Stop_Show 3324.05 BOOL  ; Stop Show
Com2_Stuur_Pomp_Hydrau_Grond 3334.01 BOOL  ; COMMUNICATIE PLC 2 NAAR PLC 1 START STUUR POMP HYDRAULIEK UNIT ARM
Com2_Stuurpomp_Hydrau_Eiland 3345.02 BOOL  ; Communicatie StuurPompen Aan Hydrualiek Eiland Plc 2 naar Plc 1
Com2_Tilt_switches_OK 3342.00 BOOL  ; Communicatie Tilt Switches OK Plc 2naar Plc 1
Com2_Uitgangs_poortjes_Dicht 3333.02 BOOL  ; Uitgangs Poortjes zijn Gesloten
Com2_Uitgangs_poortjes_Open 3333.01 BOOL  ; Uitgangs Poortjes zijn Open
Com2_VRIJGAVE_HYDRAU_ARM 3334.00 BOOL  ; COMMUNICATIE PLC 2 NAAR PLC 1 VRIJGAVE HYDRAULIEK UNIT ARM
Com2_Verhinder_Start_Show 3324.06 BOOL  ; Verhinder de Start van de Show
Com2_Vrijgave_Arm_Beweging 3337.00 BOOL
Com2_Vrijgave_Eiland_Poortjes 3344.01 BOOL  ; Communicatie Vrijgave Eiland Poortjes Plc 2 naar Plc 1
Com2_Vrijgave_Ingangs_Poortjes 3332.00 BOOL
Com2_Vrijgave_Poortjes_OK 3321.00 BOOL  ; Communicatie Vrijgave Poortjes OK Plc 2 naar Plc 1
Com2_Vrijgave_Rem_1_2_3_4 3347.11 BOOL
Com2_Vrijgave_Rotatie_Rechtsom 3347.07 BOOL
Com2_Vrijgave_Rotatie_linksom 3347.03 BOOL
Com2_Vrijgave_Show 3324.00 BOOL
Com2_Vrijgave_Tourniquets 3321.01 BOOL  ; communicatie Vrijgave Tourniquets OK Plc 2 naar Plc 1
Com3_stop_show_eiland 3600.03 BOOL  ; com 3 drukknop afbreken
DELAY_ARM_START 0141 NUMBER  ; DELAY ARM START
DFACTOR_RANGE0 D2860 CHANNEL  ; FACTOR SNELH > kLEPSTAND RANGE 0 OMLAAG
DFACTOR_RANGE0_omhoog D2850 CHANNEL  ; FACTOR SNELH > KLEPSTAND RANGE 0 Omhoog
DFACTOR_RANGE2_10 D2854 CHANNEL  ; FACTOR SNELH > KLEPSTAND RANGE 2 & 10
DFACTOR_RANGE2_omhoog D2852 CHANNEL  ; FACTOR SNELH > KLEPSTAND RANGE 2 OMHOOG
DFACTOR_RANGE4_12 D2858 REAL  ; FACTOR SNELH > KLEPSTAND RANGE 4 & 12
DFACTOR_RANGE6 D2856 CHANNEL  ; FACTOR SNELH > KLEPSTAND RANGE 3 & 11
DFACTOR_RANGE6_14 D2862 CHANNEL  ; FACTOR SNELH > KLEPSTAND RANGE 6 & 14
DFACTOR_RANGE7_15 D2864 CHANNEL  ; FACTOR SNELH > KLEPSTAND RANGE 7 & 15
DHELP_4_CNT5 D5199 INT  ; HULP ANALOOG
DHELP_5_CNT5 D5200 REAL  ; HULP ANALOOG ARM BESTURING
DIFF_FLT_PLC1 D3182 REAL  ; VERSCHIL SOLL-IST IN REAL
DSNELH_HAND D2829 INT  ; ARM SNELHEID HAND / SERVICE
DSNELH_RANGE0 D2830 INT  ; WENS SNELHEID RANGE 0
DSNELH_RANGE1 D2831 INT  ; WENS SNELHEID RANGE 1
DSNELH_RANGE10 D2840 INT  ; WENS SNELHEID RANGE 10
DSNELH_RANGE11 D2841 INT  ; WENS SNELHEID RANGE11
DSNELH_RANGE12 D2842 INT  ; WENS SNELHEID RANGE 12
DSNELH_RANGE13 D2843 INT  ; WENS SNELHEID RANGE13
DSNELH_RANGE14 D2844 INT  ; WENS SNELHEID RANGE 14
DSNELH_RANGE15 D2845 INT  ; WENS SNELHEID RANGE15
DSNELH_RANGE2 D2832 INT  ; WENS SNELHEID RANGE2
DSNELH_RANGE3 D2833 INT  ; WENS SNELHEID RANGE 3
DSNELH_RANGE4 D2834 INT  ; WENS SNELHEID RANGE 4
DSNELH_RANGE5 D2835 INT  ; WENS SNELHEID RANGE 5
DSNELH_RANGE6 D2836 INT  ; WENS SNELHEID RANGE 6
DSNELH_RANGE7 D2837 INT  ; WENS SNELHEID RANGE 7
DSNELH_RANGE8 D2838 INT  ; WENS SNELHEID RANGE8
DSNELH_RANGE9 D2839 INT  ; WENS SNELHEID RANGE9
DW_AKTIEVE_ALARMEN D35 CHANNEL
DW_Alarmen_H104 H104 CHANNEL
DW_Alarmen_H105 H105 CHANNEL
DW_Alarmen_H118 H118 CHANNEL
DW_Alarmen_H119 H119 CHANNEL
DW_Alarmen_H120 H120 UINT
DW_Alarmen_H121 H121 UINT
DW_Alarmen_H184 H184 UINT
DW_Alarmen_H185 H185 UINT
DW_Alarmen_H188 H188 CHANNEL
DW_Alarmen_H189 H189 CHANNEL
DW_Alarmen_H190 H190 CHANNEL  ; ALARMEN HYDRAU EILAND 1440-1455
DW_Alarmen_H191 H191 CHANNEL  ; ALARMEN HYDRAU EILAND 1456-1471
DW_Alarmen_H192 H192 CHANNEL
DW_Alarmen_H193 H193 CHANNEL
DW_Alarmen_H194 H194 CHANNEL
DW_Alarmen_H195 H195 CHANNEL
D_182 D182 INT
D_183 D183 CHANNEL
D_ABS_HELP2 D136 REAL  ; HELP ABS ENCODER
D_ABS_HELP3 D138 REAL  ; HELP ABS ENCODER
D_ACT_POS_ARM_PLC1 D3179 INT  ; ACT POSITIE ARM
D_ACT_POS_ARM_PLC2 D3479 INT  ; ACT POSITIE ARM
D_AFBOUW_OMHOOG D2873 INT  ; AFBOUW SNELHEID OMHOOG
D_AFBOUW_OMLAAG D2874 INT  ; AFBOUW SNELHEID OMLAAG
D_ANALOOG_UIT D189 CHANNEL  ; ANALOGE SPANNING VAN BEIDE PLC'S
D_ANA_ARM_PLC1 D3181 INT  ; ANALOGE SPANNING NAAR ARM PLC 1
D_ANA_ARM_PLC2 D3481 INT  ; SPANNING ANALOOG VAN PLC 2
D_ANA_UIT_ENAB D1400 CHANNEL  ; ENABLE CHANNEL ANALOG UIT
D_ANA_UIT_HULP D180 INT  ; HULP ANALOOG MIDDELEN
D_BOVENTIJD D2890 UINT_BCD  ; WACHTIJD BOVEN
D_CNT4_LOWER D201 INT  ; LOWER LIMIT HOEK EILAND
D_CNT4_UPPER D200 INT
D_DIFF_FLT_PLC1 D3184 REAL  ; VERSCHIL SOLL-IST IN REAL
D_DIFF_POS_PLC1 D3180 INT  ; VERSCHIL SOLL-IST PLC 1
D_DIFF_POS_PLC2 D3480 INT  ; VERSCHIL SOLL-IST  PLC 2
D_ENCODE12_GEM D193 INT  ; GEMIDDELDE COUNTER 1 & 2
D_ENCODE1_DIFF D145 INT  ; HOEK VERSCHIL ENCODER 1
D_ENCODE1_OLD D144 INT  ; HOEK OLD ENCODER 1
D_ENCODE1_PLC1 D3125 INT  ; GRADEN GETAL ENCODER 1
D_ENCODE1_PLC2 D3425 INT  ; GRADEN GETAL ENCODER 1
D_ENCODE2_DIFF D147 INT  ; HOEK VERSCHIL ENCODER 2
D_ENCODE2_OLD D146 INT  ; HOEK OLD ENCODER 2
D_ENCODE2_PLC1 D3130 INT  ; GRADEN GETAL ENCODER 2
D_ENCODE2_PLC2 D3430 INT  ; GRADEN GETAL ENCODER 2
D_ENCODE3_DIFF D149 INT  ; HOEK VERSCHIL ENCODER 3
D_ENCODE3_OLD D148 INT  ; HOEK OLD ENCODER 3
D_ENCODE3_PLC1 D3135 INT  ; GRADEN ABS ENCODER 3
D_ENCODE3_PLC2 D3435 INT  ; ENCODER 3 PLC 2
D_ENCODE4_HLP D192 INT  ; HELP COUNTER 4
D_ENCODE4_PLC1 D3190 INT  ; GRADEN GETAL ENCODER 4
D_ENCODE5 D3196 INT  ; HOEK HORIZON PLC 1
D_ENCODE5_PLC1 D3195 INT  ; HOEK HORIZON PLC 1
D_ENC_1_MIN_AFW D140 INT  ; ENCODER 1 GETAL - AFWIJKING
D_ENC_1_PLUS_AFW D139 INT  ; ENCODER 1 + AFWIJKING
D_ENC_DIFF D2872 INT  ; MAX AFWIJKING IN PULSEN
D_ENC_MAX_DOWN D2871 INT  ; MAX DAAL SNELHEID IN PULSEN
D_ENC_MAX_UP D2870 INT  ; MAX SNELHEID HOEK VERDRAAIINGOMHOOG
D_ENC_MIN_A D141 INT  ; ONDER GETAL ENCODER
D_ENC_MIN_B D143 INT  ; ENCODER MIN AFWIJKING
D_ENC_PLUS_B D142 INT  ; GETAL ENCODE PLUS AFWIJKING B
D_FACTOR D2820 REAL  ; FACTOR PULS NAAR HOEK
D_FACTOR_4 D5185 REAL  ; FACTOR PULS NAAR HOEK
D_FACTOR_5 D5191 REAL  ; FACTOR KUNSTMATIGE HORIZON
D_FACTOR_PLC1 D3177 CHANNEL  ; FACTOR TBV ARM PLC 1
D_FACTOR_PLC2 D3477 REAL  ; FACTOR TBV ARM PLC 2
D_FACTOR_abs D2822 REAL  ; FACTOR PULS NAAR HOEK abs encoder
D_HELP1 D5003 REAL
D_HELP1_ABS D5136 REAL  ; HELP ABS PULS > GRADEN
D_HELP1_CNT D150 REAL
D_HELP1_CNT1 D127 REAL  ; HULP HOEK NAAR GRADEN
D_HELP1_CNT2 D132 REAL
D_HELP1_CNT4 D187 INT  ; HULP HOEK NAAR GRADEN
D_HELP1_CNT5 D5193 REAL  ; HULP ANALOOG NAAR GRADEN
D_HELP2 D5005 REAL
D_HELP2_ABS D5138 REAL
D_HELP2_CNT D152 REAL  ; HULP HOEK NAAR GRADEN
D_HELP2_CNT1 D5128 REAL
D_HELP2_CNT2 D5129 REAL
D_HELP2_CNT4 D188 INT  ; HULP HOEK NAAR GRADEN
D_HELP2_CNT5 D5195 REAL  ; HULP ANALOOG NAAR GRADEN
D_HELP3_CNT1 D106 REAL  ; hulp bcd naar binair
D_HELP3_CNT5 D5197 INT  ; HELP 0 HORIZON
D_HELP4_CNT1 D125 INT  ; HELP INCR ENCODER
D_HELP4_CNT2 D130 INT  ; hulp bcd naar binair
D_HELP4_CNT4 D185 INT
D_HELP5_CNT1 D126 INT
D_HELP5_CNT2 D131 DINT
D_HELP5_CNT4 D186 INT
D_HELP_ANA2 D184 INT  ; HULP ANALOOG
D_HELP_DIFF D181 INT  ; HULP VERSCHIL DIFF IST--SOLL
D_HOLD_ANA_UIT D1402 CHANNEL  ; HOLD FUNCTION ANALOG UIT CHAN 1
D_INPUT D5000 INT
D_LIMIT_RANGE0 D2875 INT  ; limIt RANGE 0
D_LIMIT_RANGE1 D2876 INT  ; limit RANGE 1
D_LIMIT_RANGE2 D2877 INT  ; limit RANGE 2
D_LIMIT_RANGE3 D2878 INT  ; limit RANGE 3
D_LIMIT_RANGE4 D2879 INT  ; limit range 4
D_LIMIT_RANGE5 D2880 INT  ; limit range 5
D_LIMIT_RANGE6 D2881 INT  ; limt range 6
D_LIMIT_RANGE7 D2882 INT  ; limit range 7
D_OFFSET D2824 INT  ; OFFSET ABS ENCODER
D_OFSET_CNT5 D3197 INT  ; OFFSET  HORIZON
D_OFSET_CNT5_PLC1 D3196 INT  ; OFFSET  HORIZON
D_OUTPUT D5002 INT
D_PLC2_ACT_POS D3479 INT  ; ACT POSITIE ARM
D_PLC2_ANA_ARM D3481 INT  ; ANALOGE SPANNING NAAR ARM PLC 2
D_PLC2_DIFF_POS D3480 INT  ; VERSCHIL SOLL-IST PLC 2
D_PLC2_ENCODE1 D3425 INT  ; GRADEN GETAL ENCODER 1
D_PLC2_ENCODE2 D3430 INT  ; GRADEN GETAL ENCODER 2
D_PLC2_ENCODE3 D3435 INT  ; GRADEN ABS ENCODER
D_PLC2_ENCODE4 D3490 INT  ; GRADEN GETAL ENCODER 4
D_PULS_ABS D135 INT  ; PULS GETAL ABSOLUUT
D_RANGE10_UP D2812 INT  ; UPPER LIMIT RANGE 10 NEERGAAND
D_RANGE11_UP D2813 INT  ; UPPER LIMIT RANGE 11 NEERGAAND
D_RANGE12_UP D2814 INT  ; UPPER LIMIT RANGE 12 NEERGAAND
D_RANGE13_UP D2815 INT  ; UPPER LIMIT RANGE 13 NEERGAAND
D_RANGE14_UP D2816 INT  ; UPPER LIMIT RANGE 14 NEERGAAND
D_RANGE8_UP D2810 INT  ; UPPER LIMIT RANGE8 NEERGAAND
D_RANGE9_UP D2811 INT  ; UPPER LIMIT RANGE 9 NEERGAAND
D_RANGE_0_UP D2801 INT  ; BOVEN GRENS RANGE 0 OPGAAND
D_RANGE_1_UP D2802 INT  ; BOVEN GRENS RANGE2 OPGAAND
D_RANGE_2_UP D2803 INT  ; BOVEN GRENS RANGE 3 OPGAAND
D_RANGE_3_UP D2804 INT  ; BOVEN GRENS RANGE 3 OPGAAND
D_RANGE_4_UP D2805 INT  ; BOVEN GRENS RANGE 4 OPGAAND
D_RANGE_5_UP D2806 INT  ; BOVEN GRENS RANGE 5 OPGAAND
D_RANGE_6_UP D2807 INT  ; BOVEN GRENS RANGE 6 OPGAAND
D_RANGE_LOW D2800 INT  ; LOWER LIMT RANGE 0 & 8
D_RANGE_UP D2808 INT  ; BOVEN GRENS RANGE 7 & 15
D_SNELH_ARM_PLC1 D3175 INT  ; SNELHEID ARM PLC 1
D_SNELH_ARM_PLC2 D3475 INT  ; SNELHEID SOLL PLC 2
D_Setpoint_1 D176 CHANNEL
D_TOURN_L_MAX D156 INT  ; MAX AANTAL TOURNIKET LINKS
D_TOURN_L_TEL D155 INT  ; TEL AANTAL TOURNIKET LINKS
D_TOURN_R_MAX D158 INT  ; MAX AANTAL TOURNIKET RECHTS
D_TOURN_R_TEL D157 INT  ; TEL AANTAL TOURNIKET RECHTS
D_WENS_POS1B D178 INT  ; WENS POSITIE ENCODER 2
D_WENS_POS_PLC1 D3176 INT  ; WENS POSITIE PLC 1
D_WENS_POS_PLC2 D3476 INT  ; WENS POSITIE PLC 2
D_help_POS_ D179 INT  ; hulp wens positie
Delay_Timer_Lamp_Test 0055 NUMBER  ; Delay Timer t.b.v. de lampen test
ENCODER_1_ACCU D3127 CHANNEL  ; ENCODER 1 ACCU
ENCODER_2_ACCU D3132 CHANNEL  ; ENCODER 2 ACCU
ENC_1_ACCU_SPEED D5500 REAL  ; ENCODER 1 ACCUMULATOR SPEED CALCULATION
ENC_1_DEGREE_OF_ARM D5410 INT  ; ENCODER 1 DEGREE OF ARM
ENC_1_DEGREE_REAL D5404 REAL  ; ENCODER 1 DEGREE OF ARM IN REAL
ENC_1_PULSES_REAL D5400 REAL  ; ENCODER 1 PULSES IN REAL
ENC_1_SCALER_DEGREE D5402 REAL  ; ENCODER 1 SCALER FOR DEGREE CALCULTION
ENC_1_SPEED_DEGREE_ABS D5510 REAL  ; ENCODER 1 SPEED RESULT IN DEGREE ABSOLUTE
ENC_1_SPEED_DEGREE_ABS_R D5520 REAL  ; ENCODER SPEED DEGREE ABSOUTE REAL
ENC_1_SPEED_RESULT_DEGREE D5502 REAL  ; ENCODER 1 SPEED RESULT IN DEGREE + AND -
H_ALARM1152 H172 CHANNEL  ; ALARM WOORD 1152 -1168
H_ALARM1190 H175 CHANNEL  ; ALARM WOORD 1190-1205
H_ALARM2_1190 H275 CHANNEL  ; ALARM WOORD 1190-1205
H_ALARM_2_1152 H272 CHANNEL  ; ALARM WOORD 1152 -1168
H_ENAB_HYDRAU_EIL W220.00 BOOL  ; ENABLE HYDRAU EILAND
H_ENAB_INGANG_INT W160.00 BOOL  ; VRIJGAVE INGANGS POORTEN
H_ENAB_INGANG_SLUIT H64.02 BOOL  ; ENABLE SLUITEN INGANGS POORTEN
H_ENAB_TOURN H62.02 BOOL  ; ENABLE TOURNIKETTEN
H_ENAB_TOURN_INT H62.00 BOOL  ; TOURNIKETTEN BEIDE VRIJGEGEVN INTERN
H_ENAB_TOURN_copy H42.02 BOOL  ; ENABLE TOURNIKETTEN
H_ENAB_UITGANG_OPEN H64.03 BOOL  ; VRIJGAVE OPENEN UITGANGS POORTEN
H_ENAB_UITGANG_SLUIT H64.04 BOOL  ; VERZOEK SLUITEN UITGANGS POORTEN
H_EXTRA_TOURN_L H62.03 BOOL  ; EXTRA TELLEN TOURNIKETTEN L
H_EXTRA_TOURN_R H62.04 BOOL  ; EXTRA TELLEN TOURNIKETTEN RECHTS
H_HELP_HYDRAU_EIL W221.15 BOOL  ; HULP HYDRAU AAN EILAND
H_HELP_HYDRAU_GROND H70.03 BOOL  ; HULP HYDRAU POMPEN AAN
H_ON_HYDRAU_ARM H70.02 BOOL  ; HYDRAULIEK POMPEN ARM AAN
H_RESET_TOURN H62.01 BOOL  ; RESET TOURNIKETTEN
H_VRIJGAVE_HYDAU_ARM H70.00 BOOL  ; VRIJGAVE HYDRAULIEK UNIT ARM PLC 1 & PLC 2
I2_11WS13 353.01 BOOL  ; WERKSCHAKELAAR AAN VOEDING FREQ.REGELAAR MOTOREN ROTATIE
I2_11WS15 352.07 BOOL  ; WERKSCHAKELAAR AAN HOOFDMOTOR HYDRAULIEK EILAND
I2_12K6 354.02 BOOL  ; THERMISTOR BEWAKING TEMP. TE HOOG HOOFDMOTOR HYDRAULIEK EILAND
I2_13K13 354.08 BOOL  ; THERMISTOR BEWAKING TEMP. TE HOOG MOTOR 3 ROTATIE EILAND
I2_13K17 354.10 BOOL  ; THERMISTOR BEWAKING TEMP. TE HOOG MOTOR 4 ROTATIE EILAND
I2_13K5 354.04 BOOL  ; THERMISTOR BEWAKING TEMP. TE HOOG MOTOR 1 ROTATIE EILAND
I2_13K9 354.06 BOOL  ; THERMISTOR BEWAKING TEMP. TE HOOG MOTOR 2 ROTATIE EILAND
I2_14K13 355.00 BOOL  ; THERMISTOR BEWAKING TEMP. TE HOOG MOTOR 7 ROTATIE EILAND
I2_14K17 355.02 BOOL  ; THERMISTOR BEWAKING TEMP. TE HOOG MOTOR 8 ROTATIE EILAND
I2_14K5 354.12 BOOL  ; THERMISTOR BEWAKING TEMP. TE HOOG MOTOR 5 ROTATIE EILAND
I2_14K9 354.14 BOOL  ; THERMISTOR BEWAKING TEMP. TE HOOG MOTOR 6 ROTATIE EILAND
I2_17K10 355.05 BOOL  ; PLC 1 EN 2 MOTORREM 1/3/5/7 BEKRACHTIGT
I2_17K12 355.06 BOOL  ; PLC 1 MOTORREM 1/3/5/7 BEKRACHTIGT
I2_18K9 356.04 BOOL  ; GEEN OVERTOERENTAL ROTATIE EILAND LINKSOM/RECHTSOM
I2_19K10 356.00 BOOL  ; TILT SWITCH 1 MAXIMALE HELLING 5 GRADEN NIET OVERSCHREDEN
I2_19K12 356.01 BOOL  ; TILT SWITCH 1 MAXIMALE HELLING 5 GRADEN NIET OVERSCHREDEN
I2_19K14 356.02 BOOL  ; TILT SWITCH 2 MAXIMALE HELLING 5 GRADEN NIET OVERSCHREDEN
I2_19K16 356.03 BOOL  ; TILT SWITCH 2 MAXIMALE HELLING 5 GRADEN NIET OVERSCHREDEN
I2_20K3 356.05 BOOL  ; NOODSTOP CIRCUIT LESSENAAR LP2 OK
I2_26K3 356.06 BOOL  ; NOODSTOP CIRCUIT REMOTE I/0 PLC 1 EN 2 (eiland) OK
I2_29K13 356.08 BOOL  ; SERVICE SCHAKELAAR TECHNISCHE DIENST (RELAIS CONTROLE)
I2_29K15 356.09 BOOL  ; SERVICE SCHAKELAAR TECHNISCHE DIENST (RELAIS CONTROLE)
I2_29K3 356.12 BOOL  ; VRIJGAVE POORTJES OEVER EN EILAND
I2_29K5 356.13 BOOL  ; VRIJGAVE POORTJES OEVER EN EILAND
I2_29K7 356.14 BOOL  ; VRIJGAVE VOEDING FREQ.REGELAAR
I2_29K9 356.15 BOOL  ; VRIJGAVE VOEDING FREQ.REGELAAR
I2_40ES12 352.04 BOOL  ; FILTER BOOSTDRUK VERVUILD HYDRAULIEK EILAND
I2_40ES14 352.05 BOOL  ; FILTER STUURPOMP VERVUILD HYDRAULIEK EILAND
I2_40LS10 352.03 BOOL  ; OLIE NIVO OK
I2_40S6 352.01 BOOL  ; STUURDRUK BEWAKING HYDRAULIEK EILAND
I2_40S8 352.02 BOOL  ; BOOSTDRUK BEWAKING HYDRAULIEK EILAND
I2_40TS16 352.06 BOOL  ; OLIE TEMPERATUUR OK
I2_41S10 352.11 BOOL  ; KRUIPSNELHEID ROTATIE LINKSOM EILAND
I2_41S12 352.12 BOOL  ; STOPPOSITIE ROTATIE LINKSOM EILAND
I2_41S14 352.13 BOOL  ; KRUIPSNELHEID ROTATIE RECHTSOM EILAND
I2_41S16 352.14 BOOL  ; STOPPOSITIE RECHTSOM DRAAIEN EILAND
I2_41S18 352.15 BOOL  ; MAXIMALE EINDPOSITIE ROTATIE LINKSOM EILAND BEREIKT
I2_41S4 352.09 BOOL  ; ONDER MELDING EILAND
I2_41S7 352.10 BOOL  ; ONDER MELDING EILAND
I2_42S10 353.03 BOOL  ; OLIELEK DETECTIE FILTER
I2_42S4 353.00 BOOL  ; MAXIMALE EINDPOSITIE ROTATIE RECHTSOM EILAND BEREIKT
I2_42S8 353.02 BOOL  ; BRANDALARM EILAND (OPTIE)
I2_43LS3 353.08 BOOL  ; STAUS SIGNAL VALVE OHE 47
I2_43LS5 353.09 BOOL  ; STATUS SIGNAL VALVE OHE 145
I2_43LS7 353.10 BOOL  ; OIL LEVEL 2
I2_45K6 356.07 BOOL  ; SERVICE SCHAKELAAR TECHNISCHE DIENST INGESCHAKELD
I2_4A1_RUN 355.04 BOOL  ; RUN KONTAKT FREQ.REGELAAR MOTOREN ROTATIE
I2_4A1_STOR 355.03 BOOL  ; STORING FREQ.REGELAAR MOTOREN ROTATIE
I2_4F12 354.09 BOOL  ; THERMISCHE FOUT MOTOR 4 ROTATIE EILAND
I2_4F16 354.11 BOOL  ; THERMISCHE FOUT MOTOR 5 ROTATIE EILAND
I2_4F2 354.03 BOOL  ; THERMISCHE FOUT MOTOR 1 ROTATIE EILAND
I2_4F5 354.05 BOOL  ; THERMISCHE FOUT MOTOR 2 ROTATIE EILAND
I2_4F9 354.07 BOOL  ; THERMISCHE FOUT MOTOR 3 ROTATIE EILAND
I2_4U5_ALM 356.11 BOOL  ; KUNSTMATIGE HORIZON EILAND ALARM
I2_4U5_PRE 356.10 BOOL  ; KUNSTMATIGE HORIZON EILAND PRE ALARM
I2_5F2 354.13 BOOL  ; THERMISCHE FOUT MOTOR 6 ROTATIE EILAND
I2_5F5 354.15 BOOL  ; THERMISCHE FOUT MOTOR 7 ROTATIE EILAND
I2_5F9 355.01 BOOL  ; THERMISCHE FOUT MOTOR 8 ROTATIE EILAND
I2_6F3 354.00 BOOL  ; THERMISCHE FOUT STUURPOMP HYDRAULIEK EILAND
I2_6F6 354.01 BOOL  ; THERMISCHE FOUT HOOFDMOTOR HYDRAULIEK EILAND
I2_6WS3 352.00 BOOL  ; WERKSCHAKELAAR AAN STUURPOMP HYDRAULIEK EILAND
I2_7F12 362.03 BOOL  ; INSTALLATIE AUTOMAAT IN 230VAC VOEDING GROEP 10
I2_7F3 362.00 BOOL  ; INSTALLATIE AUTOMAAT IN 230VAC VOEDING GROEP 5
I2_7F5 362.01 BOOL  ; INSTALLATIE AUTOMAAT IN 230VAC VOEDING GROEP 6
I2_7F7 362.02 BOOL  ; INSTALLATIE AUTOMAAT IN 230VAC VOEDING GROEP 7
I2_8F11 362.05 BOOL  ; INSTALLATIE AUTOMAAT IN 24VDC VOEDING GROEP 6
I2_8F14 362.06 BOOL  ; INSTALLATIE AUTOMAAT IN 24VDC VOEDING GROEP 4
I2_8F17 362.07 BOOL  ; INSTALLATIE AUTOMAAT IN 24VDC VOEDING VRIJGAVE POORTJES
I2_8F3 362.04 BOOL  ; INSTALLATIE AUTOMAAT IN 24VDC VOEDING GROEP 5.1 T/M 5.3
I2_CNT4_OPERATE 365.07 BOOL  ; OPERATING STATUS CNT 4
I2_PF_VALVE_145 353.05 BOOL  ; POWER FEEDBACK VALVE 145
I2_PF_VALVE_47 352.08 BOOL  ; POWER FEEDBACK VALVE 47
I2_RES35304 353.04 BOOL  ; RESERVE INGANG
I2_RES35306 353.06 BOOL  ; RESERVE INGANG
I2_RES35307 353.07 BOOL  ; RESERVE INGANG
I2_RES35308 353.08 BOOL  ; RESERVE INGANG
I2_RES35309 353.09 BOOL  ; RESERVE INGANG
I2_RES35310 353.10 BOOL  ; RESERVE INGANG
I2_RES35311 353.11 BOOL  ; RESERVE INGANG
I2_RES35312 353.12 BOOL  ; RESERVE INGANG
I2_RES35313 353.13 BOOL  ; RESERVE INGANG
I2_RES35314 353.14 BOOL  ; RESERVE INGANG
I2_RES35315 353.15 BOOL  ; RESERVE INGANG
I2_RES35507 355.07 BOOL  ; RESERVE INGANG
I2_RES35508 355.08 BOOL  ; RESERVE INGANG
I2_RES35509 355.09 BOOL  ; RESERVE INGANG
I2_RES35510 355.10 BOOL  ; RESERVE INGANG
I2_RES35511 355.11 BOOL  ; RESERVE INGANG
I2_RES35512 355.12 BOOL  ; RESERVE INGANG
I2_RES35513 355.13 BOOL  ; RESERVE INGANG
I2_RES35514 355.14 BOOL  ; RESERVE INGANG
I2_RES35515 355.15 BOOL  ; RESERVE INGANG
I2_RES36208 362.08 BOOL  ; RESERVE INGANG
I2_RES36209 362.09 BOOL  ; RESERVE INGANG
I2_RES36210 362.10 BOOL  ; RESERVE INGANG
I2_RES36211 362.11 BOOL  ; RESERVE INGANG
I2_RES36212 362.12 BOOL  ; RESERVE INGANG
I2_RES36213 362.13 BOOL  ; RESERVE INGANG
I2_RES36214 362.14 BOOL  ; RESERVE INGANG
I2_RES36215 362.15 BOOL  ; RESERVE INGANG
I_11Q08 1.13 BOOL  ; AUX. CONTACT MAIN MOTOR SWITCH HYDRAULIK PUMP
I_11Q10 1.10 BOOL  ; AUX. CONTACT START MOTOR SWITCH HYDRAULIK PUMP
I_11Q12 1.11 BOOL  ; AUX. CONTACT DELTA MOTOR SWITCH HYDRAULIK PUMP
I_11WS4 0.03 BOOL  ; WERKSCHAKELAAR AAN HOOFDMOTOR HYDRAULIEK ARM
I_12K3 5.09 BOOL  ; VRIJGAVE OEVER POORTJES OPENEN
I_12K5 5.10 BOOL  ; VRIJGAVE OEVER POORTJES OPENEN
I_13Y3 4.06 BOOL  ; TERUGMELDING ONTGRENDELEN TOURNIQUET LINKS
I_13Y5 4.07 BOOL  ; TERUGMELDING ONTGRENDELEN TOURNIQUET RECHTS
I_14U2 0.05 BOOL  ; THERMISTOR BEWAKING TEMP. TE HOOG HOOFDMOTOR HYDRAULIEK ARM
I_15U2 1.09 BOOL  ; ALARM PROPORTIONELE KLEP ARM
I_18K14 3.03 BOOL  ; POORTJES EILAND GESLOTEN EN VERGRENDELD VEILIGHEIDSCIRCUIT OK (VERTRAAGD)
I_18K3 3.02 BOOL  ; POORTJES EILAND GESLOTEN EN VERGRENDELD VEILIGHEIDSCIRCUIT OK (DIRECT)
I_19K3 3.13 BOOL  ; GEEN ONDERSPANNING GEDETECTEERD
I_19K5 3.14 BOOL  ; GEEN OVERSPANNING GEDETECTEERD
I_19K7_9 1.15 BOOL  ; POORTJES EILAND GESLOTEN
I_20K3 3.04 BOOL  ; NOODSTOP CIRCUIT KAST OK
I_21K3 3.05 BOOL  ; NOODSTOP CIRCUIT LESSENAAR LP1 OK
I_22K3 3.06 BOOL  ; NOODSTOP CIRCUIT PUT CONTRAGEWICHT OK
I_23K3 3.07 BOOL  ; NOODSTOP CIRCUIT PUT EILAND OK
I_24K3 3.08 BOOL  ; NOODSTOP CIRCUIT HYDRAULIEKRUIMTE OK
I_24VOLT 5.08 BOOL  ; 24 V DC DETECTIE T.B.V. MELDING SPANNINGSUITVAL CONTROLE
I_25K3 3.09 BOOL  ; NOODSTOP CIRCUIT KONTAKTSLOT NOODBERGING OK
I_26K3 3.10 BOOL  ; NOODSTOP CIRCUIT PLC 1 EN 2 OK
I_27S12 2.09 BOOL  ; RESET NOODSTOP
I_28K15 4.15 BOOL  ; WATCHDOG PLC 2
I_28K3 3.11 BOOL  ; NOODSTOP VERZAMEL CIRCUIT DIRECT SCHAKELEND OK
I_28K7 3.12 BOOL  ; NOODSTOP VERZAMEL CIRCUIT VERTRAAGD SCHAKELEND OK
I_29K3 4.14 BOOL  ; MAXIMALE EINDBEWAKING CONTRAGEWICHT EILAND NIET BEDIEND
I_3K7 3.15 BOOL  ; KORTSLUITING OF OVERBELASTING DETECTIE VAN HOOFDSCHAKELAAR
I_40LS18 0.08 BOOL  ; OLIE NIVEAU OK
I_40PS14 0.06 BOOL  ; VOORALARM THEMPERATUUR OLIE TE HOOG OLIEKOELER
I_40PS16 0.07 BOOL  ; THEMPERATUUR OLIE OK
I_40PS6 0.02 BOOL  ; BOOSTDRUK AANWEZIG HYDRAULIEK ARM
I_41ES2 0.09 BOOL  ; FILTER BOOSTDRUK VERVUILD HYDRAULIEK ARM
I_41ES4 0.10 BOOL  ; FILTER STUURPOMP VERVUILD HYDRAULIEK ARM
I_42PS4 1.01 BOOL  ; DRUKMETING EILAND BENEDEN OP POSITIE (100 BAR)
I_42S10 1.04 BOOL  ; EILAND OP POSITIE BENEDEN
I_42S12 1.05 BOOL  ; TELPULS TOURNIQUET LINKS
I_42S14 1.06 BOOL  ; TELPULS TOURNIQUET RECHTS
I_42S6 1.02 BOOL  ; OLIE LEKDETECTIE FILTER
I_42S8 1.03 BOOL  ; EILAND OP KRUIP POSITIE BENEDEN
I_43S12 1.14 BOOL  ; POORTJE UITGANG GESLOTEN (OEVER)
I_44S2 2.00 BOOL  ; STUURSPANNING IN
I_44S6 2.02 BOOL  ; RESET ZOEMER
I_44SH10 2.04 BOOL  ; START/STOP SHOW (TOGGLE)
I_44SH12 2.05 BOOL  ; OPENEN/SLUITEN LINKER INGANGS POORTJES OEVER  (TOGGLE)
I_44SH14 2.06 BOOL  ; OPENEN/SLUITEN RECHTER INGANGS POORTJES OEVER  (TOGGLE)
I_44SH16 2.07 BOOL  ; VRIJGAVE TOURNIQUET LINKS (+ EXTRA PERSOON)
I_44SH4 2.01 BOOL  ; RESET ALGEMEEN ALARM
I_44SH8 2.03 BOOL  ; START/STOP POMPEN (TOGGLE)
I_45S15_A 3.00 BOOL  ; SERVICE SCHAKELAAR TECHNISCHE DIENST
I_45S15_B 3.01 BOOL  ; SERVICE SCHAKELAAR TECHNISCHE DIENST
I_45S5_AUTO 2.11 BOOL  ; AUTOMATISCH BEDRIJF
I_45S5_HAND 2.10 BOOL  ; HANDMATIG BEDRIJF
I_45SH11 2.13 BOOL  ; HANDBEDIENING ARM (EILAND) OMLAAG/STOP
I_45SH13 2.14 BOOL  ; HANDBEDIENING EILAND ROTATIE LINKSOM/STOP
I_45SH15 2.15 BOOL  ; HANDBEDIENING EILAND ROTATIE RECHTSOM/STOP
I_45SH2 2.08 BOOL  ; VRIJGAVE TOURNIQUET RECHTS (+ EXTRA PERSOON)
I_45SH9 2.12 BOOL  ; HANDBEDIENING ARM (EILAND) OMHOOG/STOP
I_5F15 0.12 BOOL  ; THERMISCHE FOUT STUURPOMP HYDRAULIEK ARM
I_5F7 0.04 BOOL  ; THERMISCHE FOUT HOOFDMOTOR HYDRAULIEK ARM
I_5WS15 0.11 BOOL  ; WERKSCHAKELAAR AAN STUURPOMP HYDRAULIEK ARM
I_5WS3 0.00 BOOL  ; WERKSCHAKELAAR AAN OLIEKOELER HYDRAULIEK UNIT ARM
I_6F3 0.14 BOOL  ; THERMISCHE FOUT SMEERTOESTEL HYDRAULIEK ARM
I_6F6 1.00 BOOL  ; THERMISCHE FOUT OLIE REINIGING HYDRAULIEK
I_6WS3 0.13 BOOL  ; WERKSCHAKELAAR AAN SMEERTOESTEL HYDRAULIEK ARM
I_6WS6 0.15 BOOL  ; WERKSCHAKELAAR AAN OLIE REINIGING HYDRAULIEK ARM
I_7F3_1 5.00 BOOL  ; INSTALLATIEAUTOMAAT IN 230 V AC VOEDING GROEP 1
I_7F5 5.01 BOOL  ; INSTALLATIEAUTOMAAT IN 230 V AC VOEDING GROEP 2 (DIRECT GESCHAKELD DOOR NOODSTOP
I_7F7 5.02 BOOL  ; INSTALLATIEAUTOMAAT IN 230 V AC VOEDING GROEP 3 (VETRAAGD AFVALLEND GESCHAKELD D
I_85Y14 4.08 BOOL  ; TERUGMELDING POORTJE RECHTS INGANG OPENEN (OEVER)
I_85Y16 4.09 BOOL  ; TERUGMELDING POORTJE RECHTS INGANG SLUITEN (OEVER)
I_85Y8_NEER 4.05 BOOL  ; TERUGMELDING ARM OMLAAG KLEP 3
I_85Y8_OP 4.02 BOOL  ; TERUGMELDING ARM OMHOOG KLEP 3
I_86Y4_NEER 4.04 BOOL  ; TERUGMELDING ARM OMLAAG KLEP 2
I_86Y4_OP 4.01 BOOL  ; TERUGMELDING ARM OMHOOG KLEP 2
I_86Y6_NEER 4.03 BOOL  ; TERUGMELDING ARM OMLAAG KLEP 1
I_86Y6_OP 4.00 BOOL  ; TERUGMELDING ARM OMHOOG KLEP 1
I_8F11 5.04 BOOL  ; INSTALLATIEAUTOMAAT IN 24 V DC VOEDING GROEP 2 (DIRECT GESCHAKELD DOOR NOODSTOP
I_8F13 5.05 BOOL  ; INSTALLATIEAUTOMAAT IN 24 V DC VOEDING GROEP 3 (DIRECT GESCHAKELD DOOR NOODSTOP
I_8F15 5.06 BOOL  ; INSTALLATIEAUTOMAAT IN 24 V DC VOEDING GROEP 4 (VETRAAGD AFVALLEND GESCHAKELD DO
I_8F3_1 5.03 BOOL  ; INSTALLATIEAUTOMAAT IN 24 V DC VOEDING GROEP 1.1/1.2/1.3
I_94U10A 1.08 BOOL  ; ALARM WINDMETER
I_94U10V 1.07 BOOL  ; VOORALARM WINDMETER
I_9F11 5.07 BOOL  ; INSTALLATIEAUTOMAAT IN 230 V AC VOEDING PC
I_ABS10 6.10 BOOL  ; ABSOLUTE ENCODER POSITIE ARM (32)
I_ABS11 6.11 BOOL  ; ABSOLUTE ENCODER POSITIE ARM (64)
I_ABS12 6.12 BOOL  ; ABSOLUTE ENCODER POSITIE ARM (128)
I_ABS13 6.13 BOOL  ; ABSOLUTE ENCODER POSITIE ARM (256)
I_ABS14 6.14 BOOL  ; ABSOLUTE ENCODER POSITIE ARM (512)
I_ABS15 6.15 BOOL  ; ABSOLUTE ENCODER POSITIE ARM (1024 MSB)
I_ABS5 6.05 BOOL  ; ABSOLUTE ENCODER POSITIE ARM (1 LSB)
I_ABS6 6.06 BOOL  ; ABSOLUTE ENCODER POSITIE ARM(1)
I_ABS7 6.07 BOOL  ; ABSOLUTE ENCODER POSITIE ARM (4)
I_ABS8 6.08 BOOL  ; ABSOLUTE ENCODER POSITIE ARM (8)
I_ABS9 6.09 BOOL  ; ABSOLUTE ENCODER POSITIE ARM (16)
I_CNT1_2_ERROR 2026.15 BOOL  ; ERROR COUNTER 1&2
I_CNT1_BUSY 2026.00 BOOL  ; COUNTER 1 BUSY
I_CNT2_BUSY 2026.06 BOOL  ; COUNTER 2 BUSY
I_F5 0.01 BOOL  ; THERMISCHE FOUT OLIEKOELER HYDRAULIEK UNIT ARM
I_HAG_BIT_00 5.11 BOOL  ; HAGENBUCH INFO LINK TOO MANY ERRORS
I_HAG_BIT_01 5.12 BOOL  ; HAGENBUCH INCLINOMETER TO STABILIZE THE ISLAND NOT OK
I_HAG_BIT_02 5.13 BOOL  ; HAGENBUCH STABLIZATION PUMP OUT OF ZERO POSITION (MUST BE ZERO POSITION WHEN INLAND IN HOME POSITION)
I_HAG_BIT_03 5.14 BOOL  ; HAGENBUCH SPARE
I_HAG_BIT_04 5.15 BOOL  ; Hoge temperatuur Technische Ruimte
I_HAG_BIT_05 4.10 BOOL  ; HAGENBUCH INFO LINK HAGENBUCH (FIBRE OPTIK) NOT AVAILABLE
I_HAG_BIT_06 4.11 BOOL  ; HAGENBUCH STABLIZATION ANGLE ERROR (NORMAL BEFORE TILT SWITCH ERROR)
I_HAG_BIT_07 4.12 BOOL  ; HAGENBUCH STABLIZATION PUMP OUT OF ZERO POSITION (MUST BE ZERO POSITION WHEN INLAND IN HOME POSITION)
I_HAG_BIT_08 4.13 BOOL  ; HAGENBUCH WATCHDOG SIGNAL
I_RES_ABS0 6.00 BOOL  ; RESERVE INGANG ABSOLUTE ENCODER
I_RES_ABS1 6.01 BOOL  ; RESERVE INGANG ABSOLUTE ENCODER
I_RES_ABS2 6.02 BOOL  ; RESERVE INGANG ABSOLUTE ENCODER
I_RES_ABS3 6.03 BOOL  ; RESERVE INGANG ABSOLUTE ENCODER
I_RES_ABS4 6.04 BOOL  ; RESERVE INGANG ABSOLUTE ENCODER
I_UPS_Fault 1.12 BOOL  ; UPS in storing of batterijbedrijf
LINK_FROM_PLC2_ALARM_1_1457 3345.05 BOOL  ; LINK FROM PLC 2 ALARM 1 1457
LINK_FROM_PLC2_ALARM_1_1458 3345.06 BOOL  ; LINK FROM PLC 2 ALARM 1 1458
LINK_FROM_PLC2_ALARM_1_1460 3345.07 BOOL  ; LINK FROM PLC 2 ALARM 1 1460
LINK_FROM_PLC2_ALARM_1_1463 3345.08 BOOL  ; LINK FROM PLC 2 ALARM 1 1463
MALM_1_960 H160.00 BOOL  ; ENCODER 1 TE SNEL OMHOOG
MALM_1_961 H160.01 BOOL  ; ENCODER 1 TE SNEL OMLAAG
MALM_1_962 H160.02 BOOL  ; ENCODER 2 TE SNEL OMHOOG
MALM_1_963 H160.03 BOOL  ; ENCODER 2 TE SNEL OMLAAG
MALM_1_964 H160.04 BOOL  ; ENCODER 3 TE SNEL OMHOOG
MALM_1_965 H160.05 BOOL  ; ENCODER 3 TE SNEL OMLAAG
MAX_RAMP_SPEED_DN D7102 REAL  ; MAX RAMP SPEED DOWN
MAX_RAMP_SPEED_UP D7100 REAL  ; MAX RAMP SPEED UP
MD_ARM_HAND W180.15 BOOL  ; M_DYN_ARM DRUKKNOP
MD_POORTJES W160.03 BOOL  ; DYN POORTJES
MRANGE0 W175.00 BOOL  ; IN RANGE 0
MRANGE1 W175.01 BOOL  ; IN RANGE 1
MRANGE10 W175.10 BOOL  ; IN RANGE 10
MRANGE11 W175.11 BOOL  ; IN RANGE 11
MRANGE12 W175.12 BOOL  ; IN RANGE 12
MRANGE13 W175.13 BOOL  ; IN RANGE 13
MRANGE14 W175.14 BOOL  ; IN RANGE 14
MRANGE15 W175.15 BOOL  ; IN RANGE 15
MRANGE2 W175.02 BOOL  ; IN RANGE 2
MRANGE3 W175.03 BOOL  ; IN RANGE 3
MRANGE4 W175.04 BOOL  ; IN RANGE 4
MRANGE5 W175.05 BOOL  ; IN RANGE 5
MRANGE6 W175.06 BOOL  ; IN RANGE 6
MRANGE7 W175.07 BOOL  ; IN RANGE 7
MRANGE8 W175.08 BOOL  ; IN RANGE 8
MRANGE9 W175.09 BOOL  ; IN RANGE 9
M_2ALARM_ENCODERS H258 CHANNEL  ; ALARMEN ENCODERS GROND 928-943
M_ABS_MIN H56.00 BOOL  ; VOLGENDE  AANWEZIGE BIT AFTREKKEN
M_AKTIEF_ALARM W35.00 BOOL  ; Er is minstens 1 Aktief Alarm
M_ALARM2_ENC4 H282 CHANNEL  ; ALARMEN ENCODER HOEK 4
M_ALARM2_HYDRAU_GROND H270 CHANNEL  ; ALARMEN  HYDRAU GROND 1120-1135
M_ALARM2_HYDRAU_GROND2 H271 CHANNEL  ; ALARM HYDRAU GROND 1136-1151
M_ALARM2_ING_GROND H266 CHANNEL  ; ALARMEN INGANGS POORTEN VASTE WERELD 1056-1071
M_ALARM2_TOURNIKET H264 CHANNEL  ; ALARMEN TOURNIKET 1024-1039
M_ALARM2_UITG_GROND H268 CHANNEL  ; ALARMEN UITGANG POORT VASTE WERELD 1088-1103
M_ALARM_1_0000 H100.00 BOOL  ; Alarm 1 - 0000 Er is minstens 1 Alarm in de File Main (Alarmen 1 - 0000 t/m 1 -  0031)
M_ALARM_1_0032 H102.00 BOOL  ; Alarm 1 - 0032 Er is minstens 1 Alarm in de Controllink (Alarmen 1 - 0032 t/m 1 -  0063)
M_ALARM_1_0064 H104.00 BOOL  ; Alarm 1 - 0064 Er is minstens 1 Alarm in de Devicenet (Alarmen 1 - 0064 t/m 1 -  0095)
M_ALARM_1_0096 H106.00 BOOL  ; Alarm 1 - 0096 Er is minstens 1 Alarm in de Data-Opslag (Alarmen 1 - 0096 t/m 1 -  0127)
M_ALARM_1_0128 H108.00 BOOL  ; Alarm 1-0128 Er is minstens 1 alarm in de I/O Controle afhandeling
M_ALARM_1_0160 H110.00 BOOL
M_ALARM_1_0161 H110.01 BOOL  ; Merker Alarm
M_ALARM_1_0162 H110.02 BOOL
M_ALARM_1_0163 H110.03 BOOL
M_ALARM_1_0164 H110.04 BOOL
M_ALARM_1_0225 H112.00 BOOL  ; Alarm 1- 0225 Er is minstens 1 alarm in de Noodstop afhandeling
M_ALARM_1_0226 H112.01 BOOL  ; Alarm 1- 0226 Noodstop Kast Groep 1 Gedrukt (20S4/20K3)
M_ALARM_1_0227 H112.02 BOOL  ; Alarm 1- 0227 Noodstop Lessenaar LP1 Gedrukt (21S4/21K3)
M_ALARM_1_0228 H112.03 BOOL  ; Alarm 1- 0228 Noodstop Contragewicht Put Gedrukt (22S4/22K3)
M_ALARM_1_0229 H112.04 BOOL  ; Alarm 1- 0229 Noodstop Eiland Put Gedrukt (23S4/23K3)
M_ALARM_1_0230 H112.05 BOOL  ; Alarm 1- 0230 Noodstop Hydroliekruimte Gedrukt (24S4/24K3)
M_ALARM_1_0231 H112.06 BOOL  ; Alarm 1- 0231 Noodstop Contact Noodberging (25S15/25K3/25K15/25K17)
M_ALARM_1_0232 H112.07 BOOL  ; Alarm 1- 0232 Noodstop Maximale Hoek Arm / Contragewicht  (29S4/29K3)
M_ALARM_1_0233 H112.08 BOOL
M_ALARM_1_0234 H112.09 BOOL
M_ALARM_1_0235 H112.10 BOOL
M_ALARM_1_0236 H112.11 BOOL
M_ALARM_1_0237 H112.12 BOOL
M_ALARM_1_0288 H118.00 BOOL  ; Alarm 1 - 0288 Er is minstens 1 Alarm in de wind meting
M_ALARM_1_0320 H120.00 BOOL  ; Alarm 1 - 320 Er is een alarm in de voedingen
M_ALARM_1_0321 H120.01 BOOL  ; Alarm 1-0321 OnderSpanning Beveiliging is Aangesproken (19K5)
M_ALARM_1_0322 H120.02 BOOL  ; Alarm 1-0322 OverSpanning Beveiliging is Aangesproken (19K5)
M_ALARM_1_0323 H120.03 BOOL  ; Alarm 1-0323 De Hoofdschakelaar is Getript (3K7)
M_ALARM_1_0324 H120.04 BOOL  ; Alarm 1-0324 Installatie Automaat (7F3) 230 V AC Voeding Groep 1
M_ALARM_1_0325 H120.05 BOOL  ; Alarm 1-0325 Installatie Automaat (7F5) 230 V AC Voeding Groep 2 (Noodstop Direct Afvallend)
M_ALARM_1_0326 H120.06 BOOL  ; Alarm 1-0326 Installatie Automaat (7F7) 230 V AC Voeding Groep 3 (Noodstop Vertraagt Afvallend)
M_ALARM_1_0327 H120.07 BOOL  ; Alarm 1-0327 Installatie Automaat (8F3) 24VDC Voeding Groep 1.1/1.2/1.3
M_ALARM_1_0328 H120.08 BOOL  ; Alarm 1-0328 Installatie Automaat (8F11) 24 V DC Voeding Groep 2 (Noodstop Direct Afvallend)
M_ALARM_1_0329 H120.09 BOOL  ; Alarm 1-0329 Installatie Automaat (8F15) 24 V DC Voeding Groep 4 (Noodstop Vertraagt Afvallend)
M_ALARM_1_0330 H120.10 BOOL  ; Alarm 1-0330 Installatie Automaat (9F11) 240 V AC Voeding (PC Voeding)
M_ALARM_1_0331 H120.11 BOOL  ; Alarm 1-0331 Installatie Automaat (7F3) Eiland 230VAC Voeding Groep 5
M_ALARM_1_0332 H120.12 BOOL  ; Alarm 1-0332 Installatie Automaat (7F5) Eiland 230VAC Voeding Groep 6
M_ALARM_1_0333 H120.13 BOOL  ; Alarm 1-0333 Installatie Automaat (7F7) Eiland 230VAC Voeding Groep 7
M_ALARM_1_0334 H120.14 BOOL  ; Alarm 1-0334 Installatie Automaat (7F12) Eiland 230VAC Voeding Groep 10
M_ALARM_1_0335 H120.15 BOOL  ; Alarm 1-0335 Installatie Automaat (8F3) Eiland 24VDC Voeding Groep 5.1 t/m 5.3
M_ALARM_1_0336 H121.00 BOOL  ; Alarm 1-0336 Installatie Automaat (8F11) Eiland 24VDC Voeding Groep6
M_ALARM_1_0337 H121.01 BOOL  ; Alarm 1-0337 Installatie Automaat (8F14) Eiland 24VDC Voeding Groep4
M_ALARM_1_0338 H121.02 BOOL  ; Alarm 1-0338 Installatie Automaat (8F17) Eiland 24VDC Voeding Vrijgave Poortjes
M_ALARM_1_1056 H166.00 BOOL
M_ALARM_1_1088 H168.00 BOOL
M_ALARM_1_1120 H170.00 BOOL  ; Alarm 1 -  Er is minstens 1 Alarm in de Hydrauliek van de Arm  (Alarmen 1 - 1120  t/m 1 - 1151)
M_ALARM_1_1184 H174.00 BOOL
M_ALARM_1_1216 H176.00 BOOL
M_ALARM_1_1248 H178.00 BOOL
M_ALARM_1_1280 H180.00 BOOL
M_ALARM_1_1312 H182.00 BOOL  ; Alarm 1 - 1312 Er is een alarm in de positie van het eiland.
M_ALARM_1_1344 H184.00 BOOL  ; Alarm 1 - 1344 Er is minstens 1 Alarm in de programma file Level Switches
M_ALARM_1_1345 H184.01 BOOL  ; Alarm 1 - 1345 Tilt Switch 1 Eiland aangesproken (19K10)
M_ALARM_1_1346 H184.02 BOOL  ; Alarm 1 - 1346 Tilt Switch 1 Eiland aangesproken (19K12)
M_ALARM_1_1347 H184.03 BOOL  ; Alarm 1 - 1347 Verschil tussen 19K10 & 19K12 Tilt Switch 1 Eiland aangesproken
M_ALARM_1_1348 H184.04 BOOL  ; Alarm 1 - 1348 Tilt Switch 2 Eiland aangesproken (19K14)
M_ALARM_1_1349 H184.05 BOOL  ; Alarm 1 - 1349 Tilt Switch 2 Eiland aangesproken (19K16)
M_ALARM_1_1350 H184.06 BOOL  ; Alarm 1 - 1350 Verschil tussen 19K14 & 19K16 Tilt Switch 2 Eiland aangesproken
M_ALARM_1_1376 H186.00 BOOL  ; Alarm 1 - 1376 Er is minstens 1 Alarm in de Poortjes van het Eiland  (Alarmen 1 - 1376 t/m 1 - 1440)
M_ALARM_1_1408 H188.00 BOOL
M_ALARM_1_1440 H190.00 BOOL  ; Alarm 1 - 1440 Er is minstens 1 Alarm in de Hydrauliek van het Eiland  (Alarmen 1 - 1441 t/m 1 - 1471)
M_ALARM_1_1441 H190.01 BOOL  ; ALARM 1-1441 Werkschakelaar Hulppomp Hydrau Eiland (6WS3)
M_ALARM_1_1442 H190.02 BOOL  ; ALARM 1-1442 Thermische Fout Hulppomp Hydrau Eiland (6F3)
M_ALARM_1_1443 H190.03 BOOL  ; ALARM  1-1443 Werkschakelaar Hoofdpomp Hydrau Eiland (11WS15)
M_ALARM_1_1444 H190.04 BOOL  ; ALARM 1-1444 Thermische Fout Hoofdpomp Hydrau Eiland (6F6)
M_ALARM_1_1445 H190.05 BOOL  ; ALARM 1-1445
M_ALARM_1_1446 H190.06 BOOL  ; ALARM 1-1446 Olie Nivo Te Laag Hydrau Eiland (40LS10)
M_ALARM_1_1447 H190.07 BOOL  ; ALARM  1-1447 Pilot pump filter full on island (40ES12)
M_ALARM_1_1448 H190.08 BOOL  ; ALARM 1-1448 Main pump filter full on island (40ES14)
M_ALARM_1_1449 H190.09 BOOL  ; ALARM 1-1449 Olie Temperatuur Te Hoog Hydrau Eiland (40S16)
M_ALARM_1_1450 H190.10 BOOL  ; ALARM 1-1450 Olie Lek Hydrau Eiland (42S10)
M_ALARM_1_1451 H190.11 BOOL  ; ALARM 1-1451 Stuurdruk Niet Aanwezig Hydrau Eiland (73Q4)
M_ALARM_1_1452 H190.12 BOOL  ; Alarm 1-0152 Stuurdruk Hydrauliek Eiland valt niet weg
M_ALARM_1_1453 H190.13 BOOL  ; ALARM 1-1453 SIGNAL STATUS VALVE 47 NOT OK
M_ALARM_1_1454 H190.14 BOOL  ; ALARM 1-1454 SIGNAL STATUS VALVE 145 NOT OK
M_ALARM_1_1455 H190.15 BOOL  ; ALARM 1-1455 OIL LEVEL 2 NOT OK
M_ALARM_1_1456 H191.00 BOOL  ; ALARM 1-1456 INFO LINK HAGENBUCH (FIBRE OPTIK) NOT AVAILABLE
M_ALARM_1_1457 H191.01 BOOL  ; ALARM 1-1457 INFO LINK HAGENBUCH TOO MANY ERRORS
M_ALARM_1_1458 H191.02 BOOL  ; ALARM 1-1458 INCLINOMETER TO STABILIZE THE ISLAND NOT OK
M_ALARM_1_1459 H191.03 BOOL  ; ALARM 1-1459 STABLIZATION ANGLE ERROR (NORMAL BEFORE TILT SWITCH ERROR)
M_ALARM_1_1460 H191.04 BOOL  ; ALARM 1-1460 STABLIZATION PUMP OUT OF ZERO POSITION (MUST BE ZERO POSITION WHEN INLAND IN HOME POSITION)
M_ALARM_1_1461 H191.05 BOOL  ; ALARM 1-1461 STABLIZATION PUMP NOT OK
M_ALARM_1_1462 H191.06 BOOL  ; ALARM 1-1462 HARDWARE WATCHDOG FROM HAGENBUCH MISSING
M_ALARM_1_1463 H191.07 BOOL  ; ALARM 1-1463 ANALOG OUTPUT FOR ISLAND CONTROL (HAGENBUCH PLC) NOT OK OR PASSIVATED
M_ALARM_1_1472 H192.00 BOOL
M_ALARM_1_1504 H194.00 BOOL  ; Alarm 1 - 1504 Er is minstens 1 Alarm in de Eiland Rotatie
M_ALARM_1_1505 H194.01 BOOL  ; Alarm 1 - 1505 Storing Frequentie Regelaar Rotatie Motoren
M_ALARM_1_1506 H194.02 BOOL  ; Alarm 1 - 1506 Thermische Fout (4F2) Rotatie Motor 1 Eiland
M_ALARM_1_1507 H194.03 BOOL  ; Alarm 1 - 1507 Thermische Fout (4F5) Rotatie Motor 2 Eiland
M_ALARM_1_1508 H194.04 BOOL  ; Alarm 1 - 1508 Thermische Fout (4F9) Rotatie Motor 3 Eiland
M_ALARM_1_1509 H194.05 BOOL  ; Alarm 1 - 1509 Thermische Fout (4F12) Rotatie Motor 4 Eiland
M_ALARM_1_1510 H194.06 BOOL  ; Alarm 1 - 1510 Thermische Fout (4F16) Rotatie Motor 5 Eiland
M_ALARM_1_1511 H194.07 BOOL  ; Alarm 1 - 1511 Thermische Fout (5F2) Rotatie Motor 6 Eiland
M_ALARM_1_1512 H194.08 BOOL  ; Alarm 1 - 1512 Thermische Fout (5F5) Rotatie Motor 7 Eiland
M_ALARM_1_1513 H194.09 BOOL  ; Alarm 1 - 1513 Thermische Fout (5F9) Rotatie Motor 8 Eiland
M_ALARM_1_1514 H194.10 BOOL  ; Alarm 1 - 1514 Thermistor Fout Motor 1 Eiland (13R3 / 13U2 / 13K5)
M_ALARM_1_1515 H194.11 BOOL  ; Alarm 1 - 1515 Thermistor Fout Motor 2 Eiland (13R7 / 13U6 / 13K9)
M_ALARM_1_1516 H194.12 BOOL  ; Alarm 1 - 1516 Thermistor Fout Motor 4 Eiland (13R15 / 13U14 / 13K17)
M_ALARM_1_1517 H194.13 BOOL  ; Alarm 1 - 1517 Thermistor Fout Motor 5 Eiland (14R3 / 14U2 / 14K5)
M_ALARM_1_1518 H194.14 BOOL  ; Alarm 1 - 1518 Thermistor Fout Motor 6 Eiland (14R7 / 14U6 / 14K9)
M_ALARM_1_1519 H194.15 BOOL  ; Alarm 1 - 1519 Thermistor Fout Motor 7 Eiland (14R11 / 14U10 / 14K13)
M_ALARM_1_1520 H195.00 BOOL  ; Alarm 1 - 1520 Thermistor Fout Motor 7 Eiland (14R11 / 14U10 / 14K13)
M_ALARM_1_1521 H195.01 BOOL  ; Alarm 1 - 1521 Thermistor Fout Motor 8 Eiland (14R15 / 14U14 / 14K17)
M_ALARM_1_1522 H195.01 BOOL  ; Alarm 1 - 1522 Overtoerental Rotatie Eiland (18K9)
M_ALARM_1_1832 H152.00 BOOL
M_ALARM_1_352 H122.00 BOOL
M_ALARM_1_384 H124.00 BOOL
M_ALARM_1_416 H126.00 BOOL
M_ALARM_1_448 H128.00 BOOL
M_ALARM_1_480 H130.00 BOOL
M_ALARM_1_512 H132.00 BOOL
M_ALARM_1_544 H134.00 BOOL
M_ALARM_1_576 H136.00 BOOL
M_ALARM_1_608 H138.00 BOOL
M_ALARM_1_640 H140.00 BOOL
M_ALARM_1_672 H142.00 BOOL
M_ALARM_1_704 H144.00 BOOL
M_ALARM_1_736 H146.00 BOOL
M_ALARM_1_768 H148.00 BOOL
M_ALARM_1_800 H150.00 BOOL
M_ALARM_1_864 H154.00 BOOL
M_ALARM_1_896 H156.00 BOOL
M_ALARM_1_928 H158.00 BOOL
M_ALARM_COUNTER H162 CHANNEL  ; ALARM IN COUNTER MUDUUL 992-107
M_ALARM_ENC4 H182 CHANNEL  ; ALARMEN ENCODER HOEK 4
M_ALARM_ENCODERS H158 CHANNEL  ; ALARMEN ENCODERS GROND 928-943
M_ALARM_HYDRAU_GROND H170 CHANNEL  ; ALARMEN  HYDRAU GROND 1120-1135
M_ALARM_HYDRAU_GROND2 H171 CHANNEL  ; ALARM HYDRAU GROND 1136-1151
M_ALARM_ING_GROND H166 CHANNEL  ; ALARMEN INGANGS POORTEN VASTE WERELD 1056-1071
M_ALARM_SNELHEDEN H160 CHANNEL  ; ALARMEN SNELHEDEN 960-975
M_ALARM_TOURNIKET H164 CHANNEL  ; ALARMEN TOURNIKET 1024-1039
M_ALARM_UITG_GROND H168 CHANNEL  ; ALARMEN UITGANG POORT VASTE WERELD 1088-1103
M_ALM1_928_ENC1 H158.01 BOOL  ; ENCODER 1 GROTER DAN ENCODER 2 & 3
M_ALM1_929_ENC1 H158.02 BOOL  ; ENCODER 1 KLEINER DAN ENCODER 2 & 3
M_ALM1_930_ENC2 H158.03 BOOL  ; ENCODER 2 GROTER DAN ENCODER 1 & 3
M_ALM1_931_ENC2 H158.04 BOOL  ; ENCODER 2 KLEINER DAN ENCODER 1 & 3
M_ALM1_933_ENC3 H158.05 BOOL  ; ENCODER 3 GROTER DAN ENCODER 1 & 2
M_ALM1_934_ENC3 H158.06 BOOL  ; ENCODER 3 KLEINER DAN ENCODER 1 & 2
M_ALM1_935_ENC1_2 H158.07 BOOL  ; ENCODER 1 GROTER DAN ENCODER 2 DRAAIEND
M_ALM1_936_ENC1_2 H158.08 BOOL  ; $?St$Bk?_#[29963] / Melding kruippositie niet binnen encoderwaarden (42S8) / $?St$Bk?_#[29963]
M_ALM2_928_ENC1 H258.00 BOOL  ; ENCODER 1 GROTER DAN ENCODER 2 & 3
M_ALM2_929_ENC1 H258.01 BOOL  ; ENCODER 1 KLEINER DAN ENCODER 2 & 3
M_ALM2_930_ENC2 H258.02 BOOL  ; ENCODER 2 GROTER DAN ENCODER 1 & 3
M_ALM2_931_ENC2 H258.03 BOOL  ; ENCODER 2 KLEINER DAN ENCODER 1 & 3
M_ALM2_933_ENC3 H258.04 BOOL  ; ENCODER 3 GROTER DAN ENCODER 1 & 2
M_ALM2_934_ENC3 H258.05 BOOL  ; ENCODER 3 KLEINER DAN ENCODER 1 & 2
M_ALM_1_1024 H164.00 BOOL  ; Alarm 1-0124 Er is minstens 1 alarm in de file Tourniquets
M_ALM_1_1025 H164.01 BOOL  ; ALARM 1-1025 TOURNIKET LINKS TELT BIJ BLOKKERING
M_ALM_1_1026 H164.02 BOOL  ; ALARM 1-1026 TOURNIKET RECHTS TELT BIJ BLOKKERING
M_ALM_1_1036 H171.00 BOOL  ; ALARM 1-1136 Olie Niveau te laag (40LS18) Hydrauliek Unit Arm
M_ALM_1_1056 H166.01 BOOL  ; ALARM 1 - 1056 Linker Ingangs Poortjes Niet Open (86Y12 / 43S8)
M_ALM_1_1057 H166.02 BOOL  ; ALARM 1 - 1057 Linker Ingangs Poortjes Niet Dicht (86Y14 / 43S8)
M_ALM_1_1058 H166.03 BOOL  ; ALARM 1 - 1058 Rechter Ingangs Poortjes Niet Open (85Y14 / 43S10)
M_ALM_1_1059 H166.04 BOOL  ; ALARM 1 - 1059 Rechter Ingangs Poortjes Niet Dicht (85Y16 / 43S10)
M_ALM_1_1088 H168.01 BOOL  ; ALARM 1-1088 UITGANGS POORT NIET OPEN
M_ALM_1_1089 H168.02 BOOL  ; ALARM 1-1089 UITGANGS POORT NIET DICHT
M_ALM_1_1121 H170.01 BOOL  ; ALARM 1-1121 WERKSCHAKELAAR (5WS15) HULPPOMP HYDRAULIEK ARM
M_ALM_1_1122 H170.02 BOOL  ; ALARM 1-1122 THERMISCH FOUT (5F15) HULPPOMP HYDRAULIEK ARM
M_ALM_1_1123 H170.03 BOOL  ; ALARM 1-1123 WERKSCHAKELAAR (11WS4) HOOFDPOMP HYDRAULIEK ARM
M_ALM_1_1124 H170.04 BOOL  ; ALARM 1-1124 THERMISCH FOUT (5F7) HOOFDPOMP HYDRAULIEK ARM
M_ALM_1_1125 H170.05 BOOL  ; ALARM 1-1125 THERMISTOR (14U2) HOOFDPOMP HYDRAULIEK ARM
M_ALM_1_1126 H170.06 BOOL  ; ALARM 1-1126 WERKSCHAKELAAR (5WS3) OLIE KOELER HYDRAULIEK ARM
M_ALM_1_1127 H170.07 BOOL  ; ALARM 1-1127 THERMISCH FOUT (F5) OLIE KOELER HYDRAULIEK ARM
M_ALM_1_1128 H170.08 BOOL  ; ALARM 1-1128 WERKSCHAKELAAR (6WS3)  SMEER TOESTEL ARM
M_ALM_1_1129 H170.09 BOOL  ; ALARM 1-1129 THERMISCHE FOUT (F5M7) SMEERTOESTEL ARM
M_ALM_1_1130 H170.10 BOOL  ; ALARM 1-1130 WERKSCHAKELAAR (6WS6) REINIGINGS SYSTEEM HYDRAULIEK UNIT ARM
M_ALM_1_1131 H170.11 BOOL  ; ALARM 1-1131 THERMISCHE FOUT (F5M7) REINIGING HYDRAULIEK UNIT ARM
M_ALM_1_1132 H170.12 BOOL  ; ALARM 1-1132 TEMPERATUUR OLIE (40PS16) TE HOOG HYDAULIEK UNIT ARM
M_ALM_1_1133 H170.13 BOOL  ; ALARM 1-1133 BOOSTER FILTER (41ES2) VERSTOPT HYDRAULIEK UNIT ARM
M_ALM_1_1134 H170.14 BOOL  ; ALARM1-1134 STUURFILTER (41ES4) VERSTOPT HYDRAULIEK UNIT ARM
M_ALM_1_1135 H170.15 BOOL  ; ALARM 1-1135 FILTER LEK DETECTIE (42S6) HYDRAULIEK UNIT ARM
M_ALM_1_1136 H171.00 BOOL  ; ALARM 1-1136 STUURDRUK NIET AANWEZIG (40PS6)
M_ALM_1_1137 H171.01 BOOL  ; ALARM 1-1137 OLIE NIVO (40LS18) HYDRAULIEK UNIT ARM
M_ALM_1_1138 H171.02 BOOL  ; ALARM 1-1138 Hydraulic main pump arm MS 11Q08 not OK
M_ALM_1_1139 H171.03 BOOL  ; ALARM 1-1139 Hydraulic main pump arm MS 11Q10 not OK
M_ALM_1_1140 H171.04 BOOL  ; ALARM 1-1140 Hydraulic main pump arm MS 11Q12 not OK
M_ALM_1_1190 H175.00 BOOL  ; Alarm 1190 Arm over speed
M_ALM_1_1191 H175.01 BOOL  ; Alarm 1191 Arm upper ramp over speed
M_ALM_1_1192 H175.02 BOOL  ; Alarm 1192 Arm lower ramp over speed
M_ALM_1_1193 H175.03 BOOL  ; THERMISCH HOOFDPOMP EILAND
M_ALM_1_1194 H175.04 BOOL  ; THERMISTOR HOOFDPOMP EILAND
M_ALM_1_1312 H182.01 BOOL  ; ALARM EILAND BUITEN RANGE 0 1-1313
M_ALM_1_1313 H182.02 BOOL  ; ALARM EILAND BUITEN RANGE 1 1-1313
M_ALM_1_1314 H182.03 BOOL  ; ALARM EILAND BUITEN RANGE 2-1314
M_ALM_1_1315 H182.04 BOOL  ; ALARM EILAND BUITEN RANGE 3 1-1315
M_ALM_1_1316 H182.05 BOOL  ; ALARM EILAND BUITEN RANGE 4-1316
M_ALM_1_1317 H182.06 BOOL  ; ALARM EILAND BUITEN RANGE 5 1-1317
M_ALM_1_1318 H182.07 BOOL  ; ALARM EILAND BUITEN RANGE 6 1-1318
M_ALM_1_1319 H182.08 BOOL  ; ALARM EILAND BUITEN RANGE 7 1-1319
M_ALM_1_992 H162.00 BOOL  ; ALARM IN COUNTER MODUUL GROND
M_ALM_2_1024 H264.00 BOOL  ; ALARM 2-1024 TOURNIKET LINKS TELT BIJ BLOKKERING
M_ALM_2_1025 H264.01 BOOL  ; ALARM 2-1025 TOURNIKET RECHTS TELT BIJ BLOKKERING
M_ALM_2_1036 H271.00 BOOL  ; ALARM STUURDRUK NIET AANWEZIG GROND
M_ALM_2_1056 H266.00 BOOL  ; ALARM-2-1056 INGANGS POORT LINKS NIET OPEN
M_ALM_2_1057 H266.01 BOOL  ; ALARM 2-1057  INGNGS POORT LINKS NIET DICHT
M_ALM_2_1058 H266.02 BOOL  ; ALARM 2-1058 INGANGS POORT RECHTS NIET OPEN
M_ALM_2_1059 H266.03 BOOL  ; ALARM 2-1059 INGANGS POORT RECHTS NIET DICHT
M_ALM_2_1088 H268.00 BOOL  ; ALARM 2-1088 UITGANGS POORT NIET OPEN
M_ALM_2_1089 H268.01 BOOL  ; ALARM 2-1089 UITGANGS POORT NIET DICHT
M_ALM_2_1120 H270.00 BOOL  ; ALARM_WERK SCHAK HULPPOMP GROND 2-1120
M_ALM_2_1121 H270.01 BOOL  ; ALARM THERMISCH HULPPOMP GROND 2-1121
M_ALM_2_1122 H270.02 BOOL  ; ALARM WERKSCHAK HOOFDPOMP GROND 2-1122
M_ALM_2_1123 H270.03 BOOL  ; ALARM THERMISCH HOOFDPOMP GROND 2-1123
M_ALM_2_1124 H270.04 BOOL  ; ALARM THERMISTOR HOOFDPOMP GROND 2-1124
M_ALM_2_1125 H270.05 BOOL  ; ALARM WERKSCHAK OLIE KOELER GROND 2-1125
M_ALM_2_1126 H270.06 BOOL  ; ALARM THERMISCH OLIE KOELER GROND 2-1126
M_ALM_2_1127 H270.07 BOOL  ; ALARM WERKSCHAK SMEER TOESTEL GROND 2-1127
M_ALM_2_1128 H270.08 BOOL  ; ALARM THERMISCH SMEER TOESTEL GROND2-1129
M_ALM_2_1129 H270.09 BOOL  ; ALARM WERKSCHAKELAAR HYDRAU REINIGINGS SYSTEEM GROND 2-1129
M_ALM_2_1130 H270.10 BOOL  ; ALARM THERMISCH HYDRAU REINIGING GROND 2-1130
M_ALM_2_1131 H270.11 BOOL  ; ALARM TEMPERATUUR OLIE TE HOOG 2-1131
M_ALM_2_1132 H270.12 BOOL  ; ALARM BOOSTER FILTER VERSTOPT GROND 2-1132
M_ALM_2_1133 H270.13 BOOL  ; ALARM STUUR FILTER VERSTOPT GROND 2-1133
M_ALM_2_1134 H270.14 BOOL  ; OLIE NIVO LAAG HYDRAU GROND
M_ALM_2_1152 H272.00 BOOL  ; ALARM PLC 2 WAARDE ACT-SOLL TE GROOT
M_ALM_2_1190 H275.00 BOOL  ; ALARM HYDRAU POMP 1
M_ALM_2_1191 H275.01 BOOL  ; ALARM THERMISCH HULPPOMP EILAND
M_ALM_2_1192 H275.02 BOOL  ; WERK SCHAK HOOFDPOMP EILAND
M_ALM_2_1193 H275.03 BOOL  ; THERMISCH HOOFDPOMP EILAND
M_ALM_2_1194 H275.04 BOOL  ; THERMISTOR HOOFDPOMP EILAND
M_ALM_2_1312 H282.00 BOOL  ; ALARM EILAND BUITEN RANGE 0 2-1313
M_ALM_2_1313 H282.01 BOOL  ; ALARM EILAND BUITEN RANGE 1 2-1313
M_ALM_2_1314 H282.02 BOOL  ; ALARM EILAND BUITEN RANGE 2-1314
M_ALM_2_1315 H282.03 BOOL  ; ALARM EILAND BUITEN RANGE 3 2-1315
M_ALM_2_1316 H282.04 BOOL  ; ALARM EILAND BUITEN RANGE 4- 2-1316
M_ALM_2_1317 H282.05 BOOL  ; ALARM EILAND BUITEN RANGE 5 2-1317
M_ALM_2_1318 H282.06 BOOL  ; ALARM EILAND BUITEN RANGE 6 2-1318
M_ALM_2_1319 H282.07 BOOL  ; ALARM EILAND BUITEN RANGE 7 2-1319
M_ARM_RUST H60.00 BOOL  ; STATUS ARM IN RUST
M_ARM_RUSTIG W140.00 BOOL  ; ARM IN RUST TBV CHECK ENCODERS MET ABS
M_ARM_SLOW H60.01 BOOL  ; ARM = LANGZAAM
M_AUTO_BEDRIJF W56.01 BOOL  ; Merker Auto Bedrijf
M_Alarm_1_0289 H118.01 BOOL  ; Alarm 1 - 0289 Wind_Meting Voor Alarm
M_Alarm_1_0290 H118.02 BOOL  ; Alarm 1 - 0290 Wind_Meting Alarm
M_Alarm_1_1525 H300.00 BOOL  ; Alarm 1-1525 Input verschil tussen Plc1 & Plc 2 Input : 0.00
M_Alarm_H100_H108 W36.00 BOOL
M_Alarm_H110_H118 W36.01 BOOL
M_Alarm_H120_H128 W36.02 BOOL
M_Alarm_H130_H138 W36.03 BOOL
M_Alarm_H140_H148 W36.04 BOOL
M_Alarm_H150_H158 W36.05 BOOL
M_Alarm_H160_H168 W36.06 BOOL
M_Alarm_H170_H178 W36.07 BOOL
M_Alarm_H180_H188 W36.08 BOOL
M_Alarm_H190_H198 W36.09 BOOL
M_Arm_Home W116.01 BOOL  ; Arm is gehhel beneden
M_Arm_Omhoog W180.01 BOOL  ; Merker Arm Omhoog Plc 1 & Plc 2
M_Arm_Omhoog_Delay 3037.11 BOOL  ; Afval vertraagde arm omhoog
M_Arm_Omlaag W180.02 BOOL  ; Merker Arm Omlaag Plc 1 & Plc 2
M_Auto_Rotatie_Rechtsom W230.02 BOOL
M_Auto_Rotatie_linksom W230.01 BOOL  ; Merker Auto Rotatie Linksom
M_Auto_Rotatie_rechtsom W234.02 BOOL
M_Delay_Arm_Omhoog W180.11 BOOL  ; Merker Delay Arm Omhoog Plc 1 & Plc 2
M_Delay_Arm_Omlaag W180.12 BOOL  ; Delay Merker Arm Omlaag Plc 1 & Plc 2
M_EIL_UITG_GESLOTEN W215.05 BOOL  ; EILAND UITGA POORTEN GESLOTEN
M_E_Stop_Niet_Gedrukt W25.00 BOOL  ; Merker Noodstop Niet gedrukt Plc 1 & Plc 2
M_Eiland_Home W116.02 BOOL  ; Het Eiland Is geheel Links- of Rechtsom Gedraaid
M_Eiland_Poortjes_Gesloten W210.05 BOOL  ; Alle Eiland Poortjes Gesloten
M_Eiland_Stab_Linksom W225.01 BOOL  ; Stabiliseer het Eiland naar Links Plc 1 & Plc 2
M_Eiland_Stab_Rechtsom W225.02 BOOL  ; Stabiliseer het Eiland naar Rechts Plc 1 & Plc 2
M_Enable_Show W116.15 BOOL  ; Enable Show
M_Enable_Stabilisatie W225.00 BOOL  ; Enable de Eiland Stabilisatie Plc 1 & Plc 2
M_Enable_Tourniquets W116.10 BOOL  ; Enable Tourniquets
M_Enable_Uitgangs_Poortjes_Oever W165.00 BOOL  ; Enable Uitgangs Poortjes Oever
M_GROND_ING_GESLOTEN W160.05 BOOL  ; GROND INGANGS POORTEN GESLOTEN
M_GROND_UITG_GESLOTEN W165.05 BOOL  ; GROND UITG GESLOTEN
M_HAND_BEDRIJF W56.00 BOOL  ; Merker Hand-Bedrijf
M_HULP_EILAND_OMLAAG W58.09 BOOL
M_HYDRAU_EILAND_INBEDRIJF W220.15 BOOL  ; Hydauliek pompen Eiland Inbedrijf
M_HYDRAU_OK W170.05 BOOL  ; ALLE HYDRAU ARM OK
M_Hardw_Watchdogs_OK W20.03 BOOL  ; Merker Hardware Watchdogs Plc 1 & Plc 2 OK
M_Hardw_Watchdogs_ON W20.04 BOOL  ; Merker Hardware Watchdogs Plc 1 & Plc 2 ON
M_Hardw_Watchdogs_Plc1_Plc2_OK W20.02 BOOL  ; Merker Hardware Watchdogs Plc 1 & Plc 2 OK
M_Hoofdpomp_Hydrau_Eiland W220.03 BOOL  ; Start Hoofdpomp Hydrauliek Eiland
M_Hoofdschk_OK W40.01 BOOL  ; Merker Hoofdschakelaar (3K7) OK (geen Kortsluiting of overbelasting) Plc 1 & Plc 2
M_Hydrauliek_Arm_Inbedrijf W170.05 BOOL  ; Hydraliek Arm Inbedrijf
M_Hydrauliek_Eiland_Inbedrijf W220.02 BOOL  ; Hydauliek Eiland Inbedrijf
M_INIT_CNT4_1 W185.00 BOOL  ; INIT COUNT MODE COUNTER
M_INIT_CNT4_2 W185.01 BOOL  ; INIT CNT 4 RESET MODE
M_INIT_CNT4_3 W185.02 BOOL  ; INIT CNT 4 DATA MODE
M_INIT_CNT4_4 W185.03 BOOL  ; INIT CNT 4 START COUNTING
M_INIT_CNT4_5 W185.04 BOOL  ; INIT CNT 4  INIT DONE COUNTING BUSY
M_INIT_CNT4_6 W185.05 BOOL  ; INIT CNT 4
M_Ingangs_Poortje_1_L_Dicht W160.02 BOOL
M_Ingangs_Poortje_1_Links_Open W160.01 BOOL
M_Ingangs_Poortjes_Gesloten W160.15 BOOL
M_Inst_Autom_7F12_Eiland_OK W40.13 BOOL  ; Merker Installatie-Automaat Eiland (7F12) OK Plc 1 & Plc 2
M_Inst_Autom_7F3_Eiland_OK W40.10 BOOL  ; Merker Installatie-Automaat Eiland (7F3) OK Plc 1 & Plc 2
M_Inst_Autom_7F3_OK W40.02 BOOL  ; Merker Installatie-Automaat (7F3) OK Plc 1 & Plc 2
M_Inst_Autom_7F5_Eiland_OK W40.11 BOOL  ; Merker Installatie-Automaat Eiland (7F5) OK Plc 1 & Plc 2
M_Inst_Autom_7F5_OK W40.03 BOOL  ; Merker Installatie-Automaat (7F5) OK Plc 1 & Plc 2
M_Inst_Autom_7F7_Eiland_OK W40.12 BOOL  ; Merker Installatie-Automaat Eiland (7F7) OK Plc 1 & Plc 2
M_Inst_Autom_7F7_OK W40.04 BOOL  ; Merker Installatie-Automaat (7F7) OK Plc 1 & Plc 2
M_Inst_Autom_8F11_Eiland_OK W40.15 BOOL  ; Merker Installatie-Automaat Eiland (8F11) OK Plc 1 & Plc 2
M_Inst_Autom_8F11_OK W40.06 BOOL  ; Merker Installatie-Automaat (8F11) OK Plc 1 & Plc 2
M_Inst_Autom_8F13_OK W40.07 BOOL  ; Merker Installatie-Automaat (8F13) OK Plc 1 & Plc 2
M_Inst_Autom_8F14_Eiland_OK W50.00 BOOL  ; Merker Installatie-Automaat Eiland (8F14) OK Plc 1 & Plc 2
M_Inst_Autom_8F15_OK W40.08 BOOL  ; Merker Installatie-Automaat (8F15) OK Plc 1 & Plc 2
M_Inst_Autom_8F17_Eiland_OK W50.01 BOOL  ; Merker Installatie-Automaat Eiland (8F17) OK Plc 1 & Plc 2
M_Inst_Autom_8F3_Eiland_OK W40.14 BOOL  ; Merker Installatie-Automaat Eiland (8F3) OK Plc 1 & Plc 2
M_Inst_Autom_8F3_OK W40.05 BOOL  ; Merker Installatie-Automaat (8F3) OK Plc 1 & Plc 2
M_Inst_Autom_9F11_OK W40.09 BOOL  ; Merker Installatie-Automaat (9F11) OK Plc 1 & Plc 2
M_LAMP_TEST W56.15 BOOL  ; Lamp test d.m.v.Reset zoemer drukknop langer dan 10 seconden ingedrukt te houden
M_LEES_ABS H56.01 BOOL  ; BIT GELEZEN ABS ENCODER
M_L_Ingangs_Poortjes_Open W160.03 BOOL  ; DYN POORTJES
M_NEW_ALARM W35.01 BOOL  ; Er is minstens 1 nieuw Alarm
M_NOODSTOP_DIRECT_OK W25.03 BOOL  ; Merker NoodStop Direct Plc 1 & Plc 2 OK
M_NOODSTOP_VERTRAAGT_OK W25.04 BOOL  ; Merker Noodstop Vertraagt Plc 1 & Plc 2 OK
M_OS_OPEN_SLUIT_L_OEVER_POORTJES W55.06 BOOL  ; Merker One Shot Open / Sluit Linker Poortjes Oever
M_OS_OPEN_SLUIT_R_OEVER_POORTJES W55.07 BOOL  ; Merker One Shot Open / Sluit Rechter Poortjes Oever
M_OS_Open_Ingangs_Poortjes_Eiland W65.01 BOOL  ; One Shot Open Ingangs Poortjes Eiland
M_OS_Open_Uitgangs_Poortjes_Eiland W65.03 BOOL  ; One Shot Open Uitgangs Poortjes Eiland
M_OS_RESET_ALARMEN W55.01 BOOL  ; Merker One Shot Reset Alarmen
M_OS_RESET_NOODSTOP W55.15 BOOL  ; Merker One Shot  Reset Noodstop
M_OS_RESET_ZOEMER W55.03 BOOL  ; Merker One Shot Reset Alarm Zoemer
M_OS_ROTEER_EILAND_LINKSOM W55.12 BOOL  ; Merker One Shot Roteer Eiland Linksom
M_OS_ROTEER_EILAND_RECHTSOM W55.13 BOOL  ; Merker One Shot Roteer Eiland Rechtsom
M_OS_START_STOP_HYDRAU W55.04 BOOL  ; Merker One Shot Start / Stop Hydrauliek Pompen
M_OS_START_STOP_SHOW W55.05 BOOL  ; Merker One Sot Start / Stop Show
M_OS_Show_Verlichting_Draaiend_Eiland W65.08 BOOL  ; One Shot Show VerlichtingDraaiend Gedeelte Eiland Aan
M_OS_Show_Verlichting_Vast_Eiland W65.07 BOOL  ; One Shot Show Verlichting Vaste Gedeelte Eiland Aan
M_OS_Sluit_Ingangs_Poortjes_Eiland W65.02 BOOL  ; One Shot Sluit Ingangs Poortjes Eiland
M_OS_Sluit_Uitgangs_Poortjes_Eiland W65.04 BOOL  ; One Shot Sluit Uitgangs Poortjes Eiland
M_OS_VRIJGAVE_LINKSE_TOURNIQUET W55.08 BOOL  ; Merker One Shot Vrijgave Linkse Tourniquet
M_OS_VRIJGAVE_RECHTSE_TOURNIQUET W55.09 BOOL  ; Merker One Shot Vrijgave Rechtse Tourniquet
M_Os_Beweeg_Eiland_Omhoog W55.10 BOOL  ; Merker One Shot Beweeg Eiland Omhoog
M_Os_Beweeg_Eiland_Omlaag W55.11 BOOL  ; Merker One Shot Beweeg Eiland Omhoog
M_Plc_NoodStops_OK W25.02 BOOL  ; Merker NoodStop Uitgangen Plc 1 & Plc 2 OK
M_Poortjes_Gesloten W116.03 BOOL  ; Alle Oever & Eiland Poortjes zijn Gesloten
M_RESET_NOODSTOP W55.14 BOOL  ; Merker Reset Noodstop
M_RESET_TOURN W110.02 BOOL  ; reset tourniket
M_Ready_For_Dispatch_Eiland W65.05 BOOL  ; Ready For Dispatch Eiland
M_Ready_To_Start_Show W116.07 BOOL  ; Ready to Start Show
M_Ready_to_Reset_E_Stop W25.01 BOOL  ; Ready om de Noodstop te Resetten Plc 1 & Plc 2
M_Reset_Dag_tellers W116.14 BOOL
M_Reset_Noodstop_Eiland W65.06 BOOL  ; Reset Noodstop Eiland
M_Rotatie_Linksom W230.04 BOOL  ; Rotatie Eiland Linksom
M_Rotatie_Rechtsom W230.08 BOOL
M_Rotatie_Snel_Linksom W230.06 BOOL
M_Rotatie_Snel_Rechtsom W230.10 BOOL
M_Rotatie_Traag_Linksom W230.05 BOOL
M_Rotatie_Traag_Rechtsom W230.09 BOOL
M_SERVICE_BEDERIJF W56.02 BOOL  ; Merker Service Bedrijf
M_SPANNINGS_BEVEILIGING_OK W40.00 BOOL  ; Communicatie Onder- OverSpannings beveiliging OK Plc 1 & Plc 2
M_STOP_CNT4 W185.15 BOOL  ; STOP COUNTING COUNTER 4
M_STUURSPANNING_IN W55.00 BOOL  ; Merker Stuur Spanning In
M_Show_Afbreken W116.04 BOOL  ; Show Afbreken
M_Show_Arm_Omhoog W116.08 BOOL  ; Show Arm Omhoog
M_Show_Arm_Omlaag W116.09 BOOL  ; Show Arm Omlaag
M_Show_Eiland_Rotatie W116.11 BOOL  ; Show Eiland Rotatie
M_Show_Eiland_Stabilisatie W116.10 BOOL  ; Show Eiland Stabilisatie
M_Show_Stap_0 W115.00 BOOL  ; Show Stap 0
M_Show_Stap_1 W115.01 BOOL  ; Show Stap 1
M_Show_Stap_10 W115.10 BOOL  ; Show Stap 10
M_Show_Stap_2 W115.02 BOOL  ; Show Stap 2
M_Show_Stap_3 W115.03 BOOL  ; Show Stap 3
M_Show_Stap_4 W115.04 BOOL  ; Show Stap 4
M_Show_Stap_5 W115.05 BOOL  ; Show Stap 5
M_Show_Stap_6 W115.06 BOOL  ; Show Stap 6
M_Show_Stap_7 W115.07 BOOL  ; Show Stap 7
M_Show_Stap_8 W115.08 BOOL  ; Show Stap 8
M_Show_Stap_8A W115.11 BOOL  ; Show Stap 8 A
M_Show_Stap_8B W115.12 BOOL  ; Show Stap 8 B
M_Show_Stap_9 W115.09 BOOL  ; Show Stap 9
M_Show_is_aktief W116.12 BOOL
M_Smeer_Toestel_Aan W116.13 BOOL
M_Softw_Watchdogs_ON W20.00 BOOL  ; Merker Software Watchdog on Plc 1 & Plc 2
M_Software_Watchdogs_OK W20.01 BOOL  ; Merker Software Watchdogs Plc 1 & Plc 2 OK
M_Start_Hydrau_Pompen_Eiland W220.01 BOOL  ; Start Hydrau Pompen Eiland Plc 1 & Plc 2
M_Stop_Show W116.05 BOOL  ; Show Stoppen
M_Testbit_0 H1.01 BOOL  ; Merker Testbit 0
M_Testbit_1 H1.00 BOOL  ; Merker Testbit 1
M_Testbit_10 H1.10 BOOL  ; Merker Testbit 10
M_Testbit_11 H1.11 BOOL  ; Merker Testbit 11
M_Testbit_12 H1.12 BOOL  ; Merker Testbit 12
M_Testbit_13 H1.13 BOOL  ; Merker Testbit 13
M_Testbit_14 H1.14 BOOL  ; Merker Testbit 14
M_Testbit_15 H1.15 BOOL  ; Merker Testbit 15
M_Testbit_2 H1.02 BOOL  ; Merker Testbit 2
M_Testbit_3 H1.03 BOOL  ; Merker Testbit 3
M_Testbit_4 H1.04 BOOL  ; Merker Testbit 4
M_Testbit_5 H1.05 BOOL  ; Merker Testbit 5
M_Testbit_6 H1.06 BOOL  ; Merker Testbit 6
M_Testbit_7 H1.07 BOOL  ; Merker Testbit 7
M_Testbit_8 H1.08 BOOL  ; Merker Testbit 8
M_Testbit_9 H1.09 BOOL  ; Merker Testbit 9
M_Tilt_Switches_OK W205.00 BOOL  ; Tilt Switches OK Plc 1 & Plc 2
M_Uitgangs_Poortjes_Gesloten W165.02 BOOL  ; Uitgangs Poortjes zijn Gesloten
M_Uitgangs_poortjes_Dicht W165.02 BOOL  ; Uitgangs Poortjes zijn Gesloten
M_Uitgangs_poortjes_Open W165.01 BOOL  ; Uitgangs Poortjes zijn Open
M_Verhinder_Start_Show W116.06 BOOL  ; Verhinder de Start van de Show
M_Vrijgave_Arm_Beweging W180.00 BOOL  ; Vrijgave Arm Mag Bewegen Plc 1 & Plc 2
M_Vrijgave_Ingangs_Poortjes W160.00 BOOL  ; VRIJGAVE INGANGS POORTEN
M_Vrijgave_Poortjes_OK W110.00 BOOL  ; Communicatie Vrijgave Poortjes OK Plc 1& Plc 2
M_Vrijgave_Rotatie_Linksom W230.03 BOOL
M_Vrijgave_Rotatie_Rechtsom W230.07 BOOL
M_Vrijgave_Show W116.00 BOOL  ; Vrijgave voor de Automatische show
M_Vrijgave_Start_Auto_Afloop W115.00 BOOL  ; Vrijgave Automatische Programma Afloop Plc 1 & Plc 2
M_Vrijgave_Tourniquets_OK W110.01 BOOL  ; Vrijgave Tourniquets OK Plc 1& Plc 2
M_alm1_942 H158.14 BOOL  ; $?St$Bk?_#[29964] / Encoder 1 geen waardeverandering bij aansturen Arm / $?St$Bk?_#[29964]
M_alm1_943 H158.15 BOOL  ; $?St$Bk?_#[29965] / Encoder 2 geen waardeverandering bij aansturen Arm / $?St$Bk?_#[29965]
PLC1_RANGE_0_1 3025.00 BOOL  ; IN RANGE 0 COUNTER 1
PLC1_RANGE_0_2 3026.00 BOOL  ; IN RANGE 0 COUNTER 2
PLC1_RANGE_10_1 3025.10 BOOL  ; IN RANGE 10 COUNTER 1
PLC1_RANGE_10_2 3026.10 BOOL  ; IN RANGE 10 COUNTER 2
PLC1_RANGE_11_1 3025.11 BOOL  ; IN RANGE 11 COUNTER 1
PLC1_RANGE_11_2 3026.11 BOOL  ; IN RANGE 11 COUNTER 2
PLC1_RANGE_12_1 3025.12 BOOL  ; IN RANGE 12 COUNTER 1
PLC1_RANGE_12_2 3026.12 BOOL  ; IN RANGE 12 COUNTER 2
PLC1_RANGE_13_1 3025.13 BOOL  ; IN RANGE 13 COUNTER 1
PLC1_RANGE_13_2 3026.13 BOOL  ; IN RANGE 13 COUNTER 2
PLC1_RANGE_14_1 3025.14 BOOL  ; IN RANGE 14 COUNTER 1
PLC1_RANGE_14_2 3026.14 BOOL  ; IN RANGE 14 COUNTER 2
PLC1_RANGE_15_1 3025.15 BOOL  ; IN RANGE 15 COUNTER 1
PLC1_RANGE_15_2 3026.15 BOOL  ; IN RANGE 15 COUNTER 2
PLC1_RANGE_1_1 3025.01 BOOL  ; IN RANGE 1 COUNTER 1
PLC1_RANGE_1_2 3026.01 BOOL  ; IN RANGE 1 COUNTER 2
PLC1_RANGE_2_1 3025.02 BOOL  ; IN RANGE 2 COUNTER 1
PLC1_RANGE_2_2 3026.02 BOOL  ; IN RANGE 2 COUNTER 2
PLC1_RANGE_3_1 3025.03 BOOL  ; IN RANGE 3 COUNTER 1
PLC1_RANGE_3_2 3026.03 BOOL  ; IN RANGE 3 COUNTER 2
PLC1_RANGE_4_1 3025.04 BOOL  ; IN RANGE 4 COUNTER 1
PLC1_RANGE_4_2 3026.04 BOOL  ; IN RANGE 4 COUNTER 2
PLC1_RANGE_5_1 3025.05 BOOL  ; IN RANGE 5 COUNTER 1
PLC1_RANGE_5_2 3026.05 BOOL  ; IN RANGE 5 COUNTER 2
PLC1_RANGE_6_1 3025.06 BOOL  ; IN RANGE 6 COUNTER 1
PLC1_RANGE_6_2 3026.06 BOOL  ; IN RANGE 6 COUNTER 2
PLC1_RANGE_7_1 3025.07 BOOL  ; IN RANGE 7 COUNTER 1
PLC1_RANGE_7_2 3026.07 BOOL  ; IN RANGE 7 COUNTER 2
PLC1_RANGE_8_1 3025.08 BOOL  ; IN RANGE 8 COUNTER 1
PLC1_RANGE_8_2 3026.08 BOOL  ; IN RANGE 8 COUNTER 2
PLC1_RANGE_9_1 3025.09 BOOL  ; IN RANGE 9 COUNTER 1
PLC1_RANGE_9_2 3026.09 BOOL  ; IN RANGE 9 COUNTER 2
PLC2_RANGE_0_1 3325.00 BOOL  ; IN RANGE 0 COUNTER 1
PLC2_RANGE_0_2 3326.00 BOOL  ; IN RANGE 0 COUNTER 2
PLC2_RANGE_10_1 3325.10 BOOL  ; IN RANGE 10 COUNTER 1
PLC2_RANGE_10_2 3326.10 BOOL  ; IN RANGE 10 COUNTER 2
PLC2_RANGE_11_1 3325.11 BOOL  ; IN RANGE 11 COUNTER 1
PLC2_RANGE_11_2 3326.11 BOOL  ; IN RANGE 11 COUNTER 2
PLC2_RANGE_12_1 3325.12 BOOL  ; IN RANGE 12 COUNTER 1
PLC2_RANGE_12_2 3326.12 BOOL  ; IN RANGE 12 COUNTER 2
PLC2_RANGE_13_1 3325.13 BOOL  ; IN RANGE 13 COUNTER 1
PLC2_RANGE_13_2 3326.13 BOOL  ; IN RANGE 13 COUNTER 2
PLC2_RANGE_14_1 3325.14 BOOL  ; IN RANGE 14 COUNTER 1
PLC2_RANGE_14_2 3326.14 BOOL  ; IN RANGE 14 COUNTER 2
PLC2_RANGE_15_1 3325.15 BOOL  ; IN RANGE 15 COUNTER 1
PLC2_RANGE_15_2 3326.15 BOOL  ; IN RANGE 15 COUNTER 2
PLC2_RANGE_1_1 3325.01 BOOL  ; IN RANGE 1 COUNTER 1
PLC2_RANGE_1_2 3326.01 BOOL  ; IN RANGE 1 COUNTER 2
PLC2_RANGE_2_1 3325.02 BOOL  ; IN RANGE 2 COUNTER 1
PLC2_RANGE_2_2 3326.02 BOOL  ; IN RANGE 2 COUNTER 2
PLC2_RANGE_3_1 3325.03 BOOL  ; IN RANGE 3 COUNTER 1
PLC2_RANGE_3_2 3326.03 BOOL  ; IN RANGE 3 COUNTER 2
PLC2_RANGE_4_1 3325.04 BOOL  ; IN RANGE 4 COUNTER 1
PLC2_RANGE_4_2 3326.04 BOOL  ; IN RANGE 4 COUNTER 2
PLC2_RANGE_5_1 3325.05 BOOL  ; IN RANGE 5 COUNTER 1
PLC2_RANGE_5_2 3326.05 BOOL  ; IN RANGE 5 COUNTER 2
PLC2_RANGE_6_1 3325.06 BOOL  ; IN RANGE 6 COUNTER 1
PLC2_RANGE_6_2 3326.06 BOOL  ; IN RANGE 6 COUNTER 2
PLC2_RANGE_7_1 3325.07 BOOL  ; IN RANGE 7 COUNTER 1
PLC2_RANGE_7_2 3326.07 BOOL  ; IN RANGE 7 COUNTER 2
PLC2_RANGE_8_1 3325.08 BOOL  ; IN RANGE 8 COUNTER 1
PLC2_RANGE_8_2 3326.08 BOOL  ; IN RANGE 8 COUNTER 2
PLC2_RANGE_9_1 3325.09 BOOL  ; IN RANGE 9 COUNTER 1
PLC2_RANGE_9_2 3326.09 BOOL  ; IN RANGE 9 COUNTER 2
PLC3_RANGE_12_1 3325.12 BOOL  ; IN RANGE 12 COUNTER 1
PLC3_RANGE_14_1 3325.14 BOOL  ; IN RANGE 14 COUNTER 1
PRESET_INC_HAG W225.05 BOOL  ; PRESET INCLINOMETER AT HAGENBUCH SYSTEM
R2_COUNTER4_H 364 INT  ; VALUE COUNTER 4 HIGH WORD
R2_COUNTER_4_L 363 INT  ; VALUE COUNTER 4 LOW WORD
R2_COUNTER_5 367 INT  ; ANALOGE SPANNING KUNSTMATIGE HORIZON
RAMP_DN_X1 D7014 REAL  ; BEGINNING OF RAMP AREA
RAMP_DN_X2 D7016 REAL  ; END OF RAMP AREA
RAMP_DN_Y1 D7010 REAL  ; MAX SPEED AT THE END OF RAMP
RAMP_DN_Y2 D7012 REAL  ; MAX SPEED AT THE BEGINNING OF RAMP
RAMP_UP_X1 D7004 REAL  ; BEGINNING OF RAMP AREA
RAMP_UP_X2 D7006 REAL  ; END OF RAMP AREA
RAMP_UP_Y1 D7000 REAL  ; MAX SPEED AT THE END OF RAMP
RAMP_UP_Y2 D7002 REAL  ; MAX SPEED AT THE BEGINNING OF RAMP
RESULT_A_DN D7074 REAL  ; RESULT A DOWN
RESULT_A_UP D7054 REAL  ; RESULT A UP
RESULT_A_X_DN D7072 REAL  ; RESULT A X DOWN
RESULT_A_X_UP D7052 REAL  ; RESULT A X UP
RESULT_A_Y_DN D7070 REAL  ; RESULT A Y DOWN
RESULT_A_Y_UP D7050 REAL  ; RESULT A Y UP
RESULT_B1_DN D7076 REAL  ; RESULT B1 DOWN
RESULT_B1_UP D7056 REAL  ; RESULT B1 UP
RESULT_B2_DN D7082 REAL  ; RESULT B2 DOWN
RESULT_B2_UP D7062 REAL  ; RESULT B2 UP
RESULT_B_DN D7078 REAL  ; RESULT B DOWN
RESULT_B_UP D7058 REAL  ; RESULT B UP
RESULT_COUNTER_01 2022 INT  ; PULS GETAL ENCODER 1
RESULT_COUNTER_02 2024 INT  ; PULS GETAL ENCODER 2
RESULT_POSITION_VAR_A_DN D7080 REAL  ; RESULT POSITION * VAR A DOWN
RESULT_POSITION_VAR_A_UP D7060 REAL  ; RESULT POSITION * VAR A UP
R_COUNTER1 2022 INT  ; PULS GETAL ENCODER 1
R_COUNTER2 2024 INT  ; PULS GETAL ENCODER 2
STOP_ARM_GOING_UP 3338.00 BOOL  ; STOP ARM GOING UP (LINK BIT FROM PLC 2)
TIMER_ENC1_FAULT 0150 NUMBER  ; TIMER ENCODER 1 FAUT
TIMER_ENC2_FAULT 0151 NUMBER  ; TIMER ENCODER 2 FAULT
T_ALARM_1_0161_SET T0022 BOOL
T_ALARM_1_0162_SET T0023 BOOL
T_ALARM_1_0164_SET T0024 BOOL
T_ALARM_1_1191 0320 NUMBER  ; Timer Alarm 1191
T_ALARM_1_1192 0321 NUMBER  ; Timer Alarm 1192
T_ALARM_1_1347 T0205 BOOL
T_ALARM_1_1347_SET 205 NUMBER
T_ALARM_1_1350 T0206 BOOL
T_ALARM_1_1350_SET 206 NUMBER
T_ALARM_1_1453 T0223 BOOL  ; ALARM 1-1453 SIGNAL STATUS VALVE 47 NOT OK
T_ALARM_1_1454 0224 NUMBER  ; ALARM 1-1454 SIGNAL STATUS VALVE 145 NOT OK
T_ALARM_1_1455 0225 NUMBER  ; ALARM 1-1455 OIL LEVEL 2 NOT OK
T_ALARM_1_1462_OFF 0231 NUMBER  ; ALARM 1-1462 HARDWARE WATCHDOG FROM HAGENBUCH MISSING TIMER OFF
T_ALARM_1_1462_ON 0230 NUMBER  ; ALARM 1-1462 HARDWARE WATCHDOG FROM HAGENBUCH MISSING TIMER ON
T_ARM_HYDRAULIC_ON 0240 NUMBER  ; TIMER ARM HYDRAULIC ON
T_EILAND_BOVEN T0115 BOOL  ; EILAND TIJD BOVEN
T_Hydr_Main_Pump_Arm_On 0194 NUMBER  ; Hydraulic main pump arm on delay timer
T_ING_L_DICHT T0161 BOOL  ; MAX TIJD SLUITEN INGANGS POORT LINKS
T_ING_L_DICHT_SET 161 NUMBER  ; MAX TIJD SLUITEN INGANGS POORT LINKS
T_ING_L_OPEN T0160 BOOL  ; TIJD OPENEN INGANGS POORTEN LINKS
T_ING_L_OPEN_SET 160 NUMBER  ; MAX TIJD OPENE INGANG LINKS
T_ING_R_DICHT T0163 BOOL  ; MAX TIJD OPENEN INGANGS POORTEN RECHTS
T_ING_R_DICHT_SET 163 NUMBER  ; MAX TIJD OPEPEN INGANGS POORTEN RECHTS
T_ING_R_OPEN T0162 BOOL  ; MAX TIJD OPENEN INGANGS POORT RECHTS
T_ING_R_OPEN_SET 162 NUMBER  ; MAX TIJD OPEPEN INGANGS POORT RECTS
T_ISLAND_HYDRAULIC_ON 0241 NUMBER  ; TIMER ISLAND HYDRAULIC ON
T_Input_0_00 500 NUMBER
T_MS_11Q08_not_OK 0195 NUMBER  ; Hydraulic main pump arm MS 11Q08 not OK
T_MS_11Q10_not_OK 0196 NUMBER  ; Hydraulic main pump arm MS 11Q10 not OK
T_MS_11Q12_not_OK 0197 NUMBER  ; Hydraulic main pump arm MS 11Q12 not OK
T_Open_Uitgangs_poortjes T0165 BOOL  ; Maximale tijd Open Uitgangs Poortjes
T_PRESET_INC_HAGENBUCH 0311 NUMBER  ; PRESET INCLINOMETER HAGENBUCH
T_RESET_HAGENBUCH 0310 NUMBER  ; TIMER RESET ERROR HAGENBUCH SYSTEM
T_SNELHEID 145 NUMBER  ; SNELHEIDS METING ARM
T_SNELHEID_ACT T0145 BOOL  ; TIMER TBV ARM SNELEHEID
T_STUURDRUK_SET_GROND 170 NUMBER  ; DELAY STUURDRUK AANWEZIG
T_STUUR_DRUK T0170 BOOL  ; DELAY STUURDRUK MOET AANWEZIG ZIJN
T_STUUR_DRUK_EIL T0220 BOOL  ; STUURDRUK AANWEZIG EILAND
T_SUURDRUK_EILAND_SET 220 NUMBER  ; DELAY STUUR DRUK AANWEZIG
T_Sluit_Uitgangs_Poortjes T0166 BOOL  ; Maximale tijd sluit uitgangs poortjes
T_UITG_DICHT T0169 BOOL  ; MAX TIJD UITGANGS POORT SLUITEN
T_UITG_DICHT_SET 169 NUMBER  ; MAX TIJD SLUITEN UITGANGS POORT
T_UITG_OPEN_SET 165 NUMBER  ; MAX TIJD OPENEN UITGANGS POORTEN
T_Watchdog_Pulse_Check_Plc_2_H T0020 BOOL
T_Watchdog_Pulse_Check_Plc_2_L T0021 BOOL
T_Watchdog_Pulse_Check_Plc_2_Set 20 NUMBER
T_Watchdog_Pulse_Check_Plc_2_Set_H 20 NUMBER
T_Watchdog_Pulse_Check_Plc_2_Set_L 21 NUMBER
T_eiland_boven 0115 NUMBER  ; eiland boven tijd
T_eilandpoort_set 164 NUMBER  ; delay eiland poortjes melding
Test_Speed D7500 REAL
Totale_Dag_Teller_Tourniquets D159 CHANNEL  ; Totale Dag teller Linker & Rechter Tournoquets
U2_72K10 60.03 BOOL  ; ENABLE LINKSOM FREQ.REGELAAR MOTOREN ROTATIE
U2_72K12 60.04 BOOL  ; VRIJGEVEN MOTORREM 1,2,3 EN 4 ROTATIE EILAND
U2_72K14 60.05 BOOL  ; BYPASS ISLAND STABILISATION PUMP VALVE 47
U2_72K16 60.06 BOOL  ; VRIJGAVE POORTJES EILAND
U2_72K18 60.07 BOOL  ; BYPASS ISLAND STABILISATION CYLINDER VALVE 145
U2_72K6 60.01 BOOL  ; VOEDING FREQ.REGELAAR MOTOREN ROTATIE
U2_72K8 60.02 BOOL  ; ENABLE RECHTSOM FREQ.REGELAAR MOTOREN ROTATIE
U2_73K6 61.02 BOOL  ; HOOFDMOTOR HYDRAULIEK EILAND
U2_73K8 61.03 BOOL  ; VRIJGAVE POORTJES EILAND
U2_73Q4 61.01 BOOL  ; STUURPOMP HYDRAULIEK EILAND
U2_ARM_DIRECTION 61.07 BOOL  ; ARM DIRECTION 1=UP / 0=DOWN
U2_CNT4_COUNT_READ 64.06 BOOL  ; READ COUNTER VALUE
U2_CNT4_COUNT_SET 64.02 BOOL  ; COUNTING SET BIT
U2_CNT4_MODE_1 64.11 BOOL  ; DIFF PHASE 1x
U2_CNT4_MODE_2 64.10 BOOL  ; DIFF PHASE 1x
U2_CNT4_MODE_3 64.12 BOOL  ; RESET MODE
U2_CNT4_MODE_4 64.13 BOOL  ; RESET MODE
U2_CNT4_MODE_5 64.14 BOOL  ; RESET MODE
U2_CNT4_MODE_7 64.03 BOOL  ; DATA MODE 0=BCD 1=HEX
U2_CNT4_RESET 64.07 BOOL  ; INTERNAL RESET
U2_E_STOP_ISLAND 61.05 BOOL  ; E-STOP SIGNAL TO HYDRAULIK UNIT ISLAND
U2_NOOD_PCL1A 60.00 BOOL  ; NOODSTOP CIRCUIT REMOTE I/O PLC1
U2_NOOD_PCL1B 61.00 BOOL  ; NOODSTOP CIRCUIT REMOTE I/O PLC1
U2_STABILISATION_ENABLE 61.06 BOOL  ; STABILISATION ENABLE ISLAND
U55K4_1 13.00 BOOL  ; WATCH DOG PLC1 NIEUW
U_55K4 8.01 BOOL  ; WATCH DOG PLC 1
U_85K10 8.04 BOOL  ; ONTGRENDELEN TOURNIQUET LINKS
U_85K12 8.05 BOOL  ; ONTGRENDELEN TOURNIQUET RECHTS
U_85Y14 8.06 BOOL  ; POORTJE RECHTS INGANG OPENEN (OEVER)
U_85Y16 8.07 BOOL  ; POORTJE RECHTS INGANG SLUITEN (OEVER)
U_85Y6 8.02 BOOL  ; ARM OMHOOG KLEP 1
U_85Y8 8.03 BOOL  ; ARM OMLAAG KLEP 1
U_86Y10 9.04 BOOL  ; ARM OMLAAG KLEP 3
U_86Y4 9.01 BOOL  ; ARM OMHOOG KLEP 2
U_86Y6 9.02 BOOL  ; ARM OMLAAG KLEP 2
U_86Y8 9.03 BOOL  ; ARM OMHOOG KLEP 3
U_87K8 10.03 BOOL  ; START HOOFDMOTOR HYDRAULIEK UNIT ARM
U_87Q10 10.04 BOOL  ; START STUURPOMP HYDRAULIEK UNIT ARM
U_87Q12 10.05 BOOL  ; START SMEERTOESTEL HYDRAULIEK UNIT ARM
U_87Q14 10.06 BOOL  ; START OLIEREINIGING HYDRAULIEK UNIT ARM
U_87Q6 10.02 BOOL  ; START OLIEKOELER HYDRAULIEK UNIT ARM
U_87Y2 10.00 BOOL  ; POORTJE UITGANG OPENEN (OEVER)
U_87Y4 10.01 BOOL  ; POORTJE UITGANG SLUITEN (OEVER)
U_ANA_ARM 2041 CHANNEL  ; ANALOOG _UIT_CHAN1 TBV ARM BESTURING
U_ENAB_ANA_CHAN1 2040.00 BOOL  ; CHAN 1 ENABLE
U_HAG_BIT_10 61.04 BOOL  ; HAGENBUCH TILT SENSOREN OK
U_HAG_PRESET 9.05 BOOL  ; HAGENBUCH PRESET INCLINOMETER
U_HAG_RESET 9.06 BOOL  ; HAGENBUCH ALARM RESET
U_NS_PLC1A 8.00 BOOL  ; NOODSTOP CIRCUIT PLC 1
U_NS_PLC1B 9.00 BOOL  ; NOODSTOP CIRCUIT PLC 1
U_Open_Ingangs_Poortje_1_Links_Oever 12.04 BOOL
U_Open_Ingangs_Poortje_1_Rechts_Oever 12.00 BOOL  ; Open Ingangs Poortje 1 Rechter zijde Oever
U_Open_Ingangs_Poortje_2_Links_Oever 12.05 BOOL
U_Open_Ingangs_Poortje_2_Rechts_Oever 12.01 BOOL  ; Open Ingangs Poortje 2 Rechter zijde Oever
U_Open_Uitgangs_Poortje_1_Oever 12.08 BOOL
U_Open_Uitgangs_Poortje_2_Oever 12.09 BOOL
U_RES907 9.07 BOOL  ; RESERVE UITGANG
U_RES_10_07 10.07 BOOL  ; RESERVE
U_Res_noodstop 9.07 BOOL  ; Mogelijk om noodstop te resetten
U_Sluit_Ingangs_Poortje_1_Links_Oever 12.06 BOOL
U_Sluit_Ingangs_Poortje_1_Rechts_Oever 12.02 BOOL
U_Sluit_Ingangs_Poortje_2_Links_Oever 12.07 BOOL
U_Sluit_Ingangs_Poortje_2_Rechts_Oever 12.03 BOOL
U_Sluit_Uitgangs_Poortje_1_Oever 12.10 BOOL
U_Sluit_Uitgangs_Poortje_2_Oever 12.11 BOOL
W_ING_PRT_EIL_GESL W210.05 BOOL  ; Ingangs Poortjes Eiland Gesloten Plc 1 & 2 & 3
W_RANGE0_CNT1 W125.00 BOOL  ; ARM IN RANGE 0
W_RANGE0_CNT2 W126.00 BOOL  ; ARM IN RANGE 0
W_RANGE0_PLC1 3036.00 BOOL  ; ARM IN RANGE 0
W_RANGE0_PLC2 3336.00 BOOL  ; ARM IN RANGE 0
W_RANGE10_CNT1 W125.10 BOOL  ; ARM IN RANGE 10
W_RANGE10_CNT2 W126.10 BOOL  ; ARM IN RANGE 10
W_RANGE10_PLC1 3036.10 BOOL  ; ARM IN RANGE 10
W_RANGE10_PLC2 3336.10 BOOL  ; ARM IN RANGE 10
W_RANGE11_CNT1 W125.11 BOOL  ; ARM IN RANGE 11
W_RANGE11_CNT2 W126.11 BOOL  ; ARM IN RANGE 11
W_RANGE11_PLC1 3036.11 BOOL  ; ARM IN RANGE 11
W_RANGE11_PLC2 3336.11 BOOL  ; ARM IN RANGE 11
W_RANGE12_CNT1 W125.12 BOOL  ; ARM IN RANGE 12
W_RANGE12_CNT2 W126.12 BOOL  ; ARM IN RANGE 12
W_RANGE12_PLC1 3036.12 BOOL  ; ARM IN RANGE 12
W_RANGE12_PLC2 3336.12 BOOL  ; ARM IN RANGE 12
W_RANGE13_CNT1 W125.13 BOOL  ; ARM IN RANGE 13
W_RANGE13_CNT2 W126.13 BOOL  ; ARM IN RANGE 13
W_RANGE13_PLC1 3036.13 BOOL  ; ARM IN RANGE 13
W_RANGE13_PLC2 3336.13 BOOL  ; ARM IN RANGE 13
W_RANGE14_CNT1 W125.14 BOOL  ; ARM IN RANGE 14
W_RANGE14_CNT2 W126.14 BOOL  ; ARM IN RANGE 14
W_RANGE14_PLC1 3036.14 BOOL  ; ARM IN RANGE 14
W_RANGE14_PLC2 3336.14 BOOL  ; ARM IN RANGE 14
W_RANGE15_CNT1 W125.15 BOOL  ; ARM IN RANGE 15
W_RANGE15_CNT2 W126.15 BOOL  ; ARM IN RANGE 15
W_RANGE15_PLC1 3036.15 BOOL  ; ARM IN RANGE 15
W_RANGE15_PLC2 3336.15 BOOL  ; ARM IN RANGE 15
W_RANGE1_CNT1 W125.01 BOOL  ; ARM IN RANGE 1
W_RANGE1_CNT2 W126.01 BOOL  ; ARM IN RANGE 1
W_RANGE1_PLC1 3036.01 BOOL  ; ARM IN RANGE 1
W_RANGE1_PLC2 3336.01 BOOL  ; ARM IN RANGE 1
W_RANGE2_CNT1 W125.02 BOOL  ; ARM IN RANGE 2
W_RANGE2_CNT2 W126.02 BOOL  ; ARM IN RANGE 2
W_RANGE2_PLC1 3036.02 BOOL  ; ARM IN RANGE 2
W_RANGE2_PLC2 3336.02 BOOL  ; ARM IN RANGE 2
W_RANGE3_CNT1 W125.03 BOOL  ; ARM IN RANGE 3
W_RANGE3_CNT2 W126.03 BOOL  ; ARM IN RANGE 3
W_RANGE3_PLC1 3036.03 BOOL  ; ARM IN RANGE 3
W_RANGE3_PLC2 3336.03 BOOL  ; ARM IN RANGE 3
W_RANGE4_CNT1 W125.04 BOOL  ; ARM IN RANGE 4
W_RANGE4_CNT2 W126.04 BOOL  ; ARM IN RANGE 4
W_RANGE4_PLC1 3036.04 BOOL  ; ARM IN RANGE 4
W_RANGE4_PLC2 3336.04 BOOL  ; ARM IN RANGE 4
W_RANGE5_CNT1 W125.05 BOOL  ; ARM IN RANGE 5
W_RANGE5_CNT2 W126.05 BOOL  ; ARM IN RANGE 5
W_RANGE5_PLC1 3036.05 BOOL  ; ARM IN RANGE 5
W_RANGE5_PLC2 3336.05 BOOL  ; ARM IN RANGE 5
W_RANGE6_CNT1 W125.06 BOOL  ; ARM IN RANGE 6
W_RANGE6_CNT2 W126.06 BOOL  ; ARM IN RANGE 6
W_RANGE6_PLC1 3036.06 BOOL  ; ARM IN RANGE 6
W_RANGE6_PLC2 3336.06 BOOL  ; ARM IN RANGE 6
W_RANGE7_CNT1 W125.07 BOOL  ; ARM IN RANGE 7
W_RANGE7_CNT2 W126.07 BOOL  ; ARM IN RANGE 7
W_RANGE7_PLC1 3036.07 BOOL  ; ARM IN RANGE 7
W_RANGE7_PLC2 3336.07 BOOL  ; ARM IN RANGE 7
W_RANGE8_CNT1 W125.08 BOOL  ; ARM IN RANGE 8
W_RANGE8_CNT2 W126.08 BOOL  ; ARM IN RANGE 8
W_RANGE8_PLC1 3036.08 BOOL  ; ARM IN RANGE 8
W_RANGE8_PLC2 3336.08 BOOL  ; ARM IN RANGE 8
W_RANGE9_CNT1 W125.09 BOOL  ; ARM IN RANGE 9
W_RANGE9_CNT2 W126.09 BOOL  ; ARM IN RANGE 9
W_RANGE9_PLC1 3036.09 BOOL  ; ARM IN RANGE 9
W_RANGE9_PLC2 3336.09 BOOL  ; ARM IN RANGE 9
com1_Eiland_Home 3024.02 BOOL  ; Het Eiland Is geheel Links- of Rechtsom Gedraaid
scada_afbreken_eiland H118.03 BOOL  ; scade-stop-eiland
scada_afbreken_grond H118.04 BOOL  ; scada-stop-grond
t_eilandpoort_act T0164 BOOL  ; edelay eiland poortjes
t_soll_diff_arm T0175 BOOL  ; tijd comm verschil soll- ist
t_soll_diff_arm_set 175 NUMBER  ; diff soll-ist waarde arm

## Program ALGEMEEN (cyclic task 0)

### Section Main

